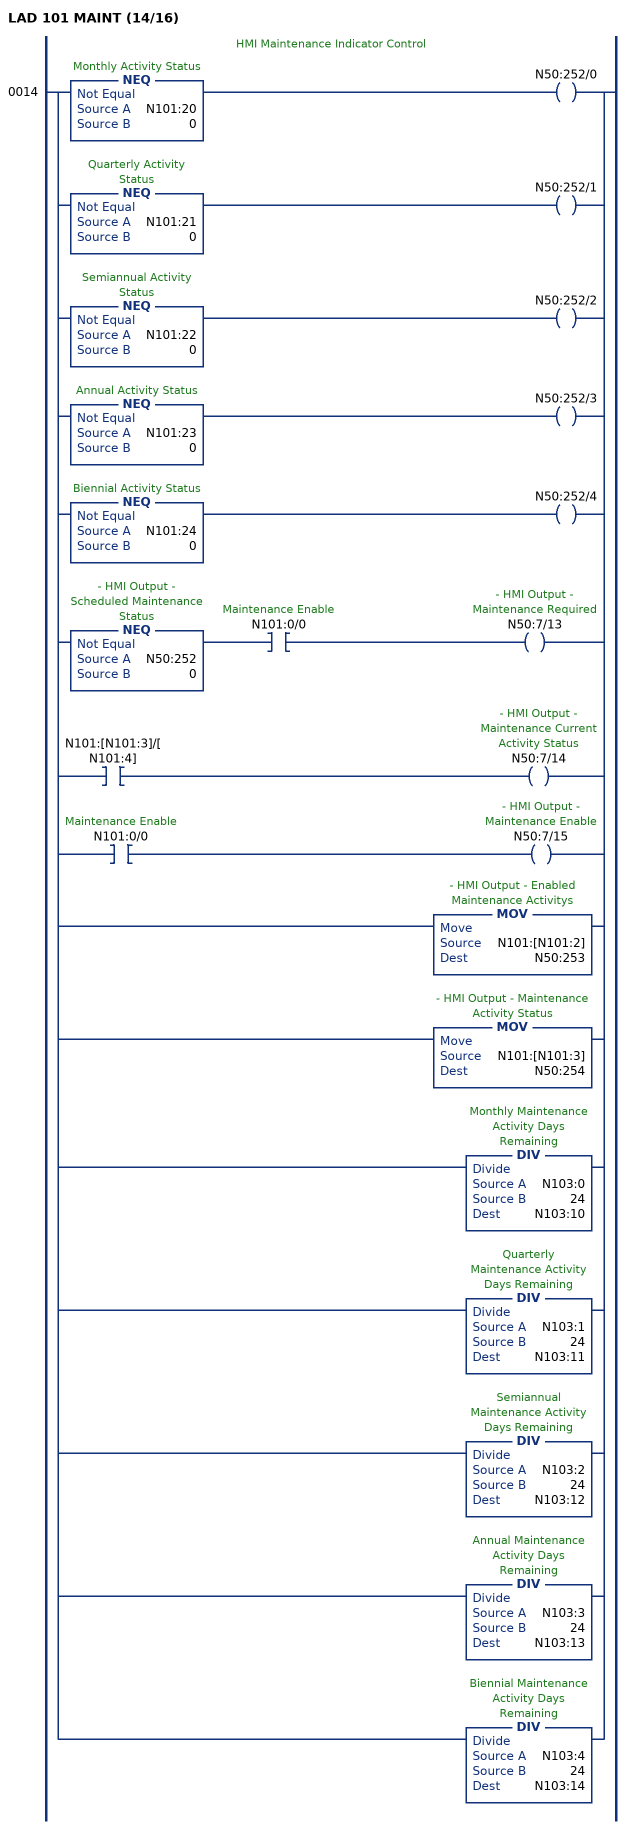
% Rung: 14 %
% HMI Maintenance Indicator Control %
SOR BST BST NEQ N101:20 0 OTE N50:252/0 NXB NEQ N101:21 0 OTE N50:252/1 NXB NEQ N101:22 0 OTE N50:252/2 NXB NEQ N101:23 0 OTE N50:252/3 NXB NEQ N101:24 0 OTE N50:252/4 NXB NEQ N50:252 0 XIC N101:0/0 OTE N50:7/13 BND NXB XIC N101:[N101:3]/[N101:4] OTE N50:7/14 NXB XIC N101:0/0 OTE N50:7/15 NXB BST MOV N101:[N101:2] N50:253 NXB MOV N101:[N101:3] N50:254 BND NXB BST DIV N103:0 24 N103:10 NXB DIV N103:1 24 N103:11 NXB DIV N103:2 24 N103:12 NXB DIV N103:3 24 N103:13 NXB DIV N103:4 24 N103:14 BND BND EOR
%   N101:20  "Monthly Activity Status" %
%   N101:21  "Quarterly Activity Status" %
%   N101:22  "Semiannual Activity Status" %
%   N101:23  "Annual Activity Status" %
%   N101:24  "Biennial Activity Status" %
%   N50:252  "- HMI Output - Scheduled Maintenance Status" %
%   N101:0/0  "Maintenance Enable" %
%   N50:7/13  "- HMI Output - Maintenance Required" %
%   N101:3  "Maintenance Schedule Index Plus 20" %
%   N101:4  "Maintenance Activity Index" %
%   N50:7/14  "- HMI Output - Maintenance Current Activity Status" %
%   N50:7/15  "- HMI Output - Maintenance Enable" %
%   N101:2  "Maintenance Schedule Index Plus 10" %
%   N50:253  "- HMI Output - Enabled Maintenance Activitys" %
%   N50:254  "- HMI Output - Maintenance Activity Status" %
%   N103:0  "Monthly Maintenance Activity Hours Remaining" %
%   N103:10  "Monthly Maintenance Activity Days Remaining" %
%   N103:1  "Quarterly Maintenance Activity Hours Remaining" %
%   N103:11  "Quarterly Maintenance Activity Days Remaining" %
%   N103:2  "Semiannual Maintenance Activity Hours Remaining" %
%   N103:12  "Semiannual Maintenance Activity Days Remaining" %
%   N103:3  "Annual Maintenance Activity Hours Remaining" %
%   N103:13  "Annual Maintenance Activity Days Remaining" %
%   N103:4  "Biennial Maintenance Activity Hours Remaining" %
%   N103:14  "Biennial Maintenance Activity Days Remaining" %

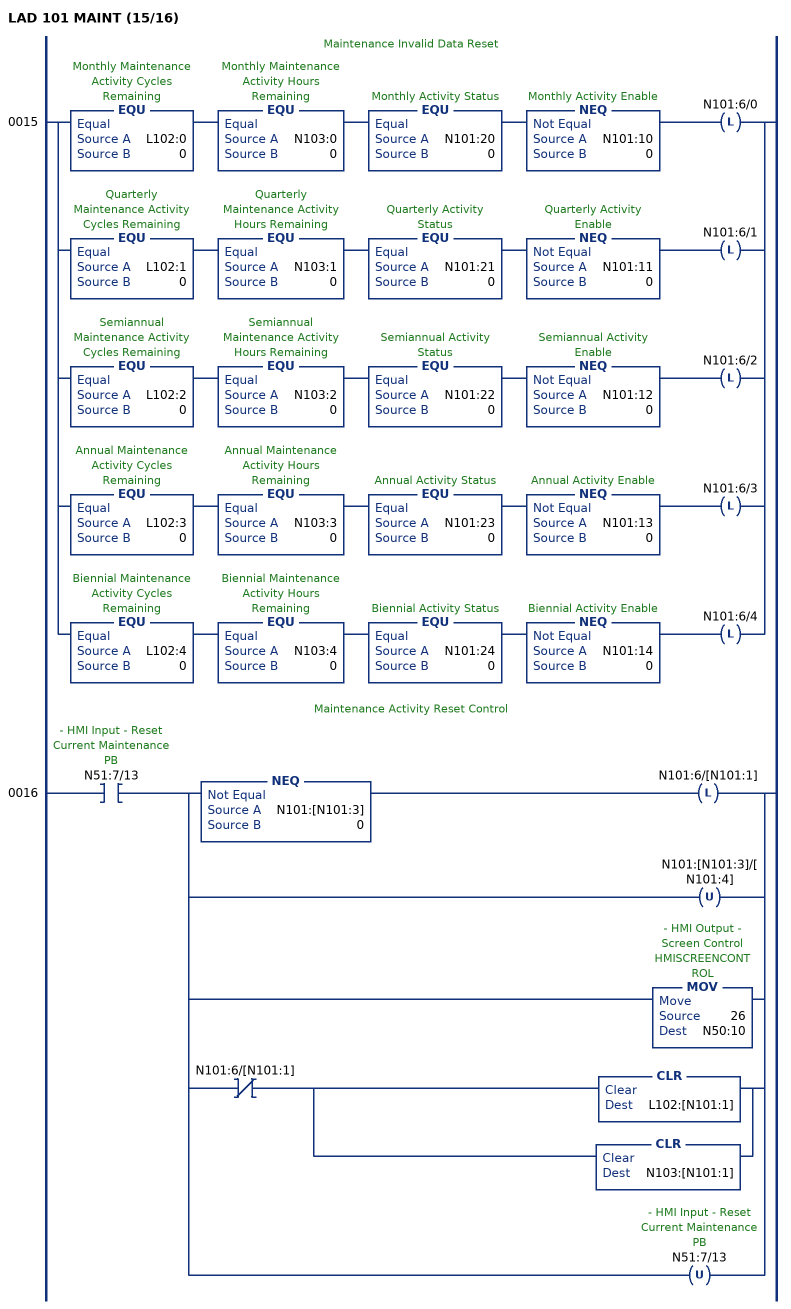
% Rung: 15 %
% Maintenance Invalid Data Reset %
SOR BST EQU L102:0 0 EQU N103:0 0 EQU N101:20 0 NEQ N101:10 0 OTL N101:6/0 NXB EQU L102:1 0 EQU N103:1 0 EQU N101:21 0 NEQ N101:11 0 OTL N101:6/1 NXB EQU L102:2 0 EQU N103:2 0 EQU N101:22 0 NEQ N101:12 0 OTL N101:6/2 NXB EQU L102:3 0 EQU N103:3 0 EQU N101:23 0 NEQ N101:13 0 OTL N101:6/3 NXB EQU L102:4 0 EQU N103:4 0 EQU N101:24 0 NEQ N101:14 0 OTL N101:6/4 BND EOR
%   L102:0  "Monthly Maintenance Activity Cycles Remaining" %
%   N103:0  "Monthly Maintenance Activity Hours Remaining" %
%   N101:20  "Monthly Activity Status" %
%   N101:10  "Monthly Activity Enable" %
%   L102:1  "Quarterly Maintenance Activity Cycles Remaining" %
%   N103:1  "Quarterly Maintenance Activity Hours Remaining" %
%   N101:21  "Quarterly Activity Status" %
%   N101:11  "Quarterly Activity Enable" %
%   L102:2  "Semiannual Maintenance Activity Cycles Remaining" %
%   N103:2  "Semiannual Maintenance Activity Hours Remaining" %
%   N101:22  "Semiannual Activity Status" %
%   N101:12  "Semiannual Activity Enable" %
%   L102:3  "Annual Maintenance Activity Cycles Remaining" %
%   N103:3  "Annual Maintenance Activity Hours Remaining" %
%   N101:23  "Annual Activity Status" %
%   N101:13  "Annual Activity Enable" %
%   L102:4  "Biennial Maintenance Activity Cycles Remaining" %
%   N103:4  "Biennial Maintenance Activity Hours Remaining" %
%   N101:24  "Biennial Activity Status" %
%   N101:14  "Biennial Activity Enable" %
% Rung: 16 %
% Maintenance Activity Reset Control %
SOR XIC N51:7/13 BST NEQ N101:[N101:3] 0 OTL N101:6/[N101:1] NXB OTU N101:[N101:3]/[N101:4] NXB MOV 26 N50:10 NXB XIO N101:6/[N101:1] BST CLR L102:[N101:1] NXB CLR N103:[N101:1] BND NXB OTU N51:7/13 BND EOR
%   N51:7/13  "- HMI Input - Reset Current Maintenance PB" %
%   N101:3  "Maintenance Schedule Index Plus 20" %
%   N101:6  "Maintenance Reset" %
%   N101:1  "Maintenance Schedule Index" %
%   N101:4  "Maintenance Activity Index" %
%   N50:10  HMISCREENCONTROL  "- HMI Output - Screen Control" %

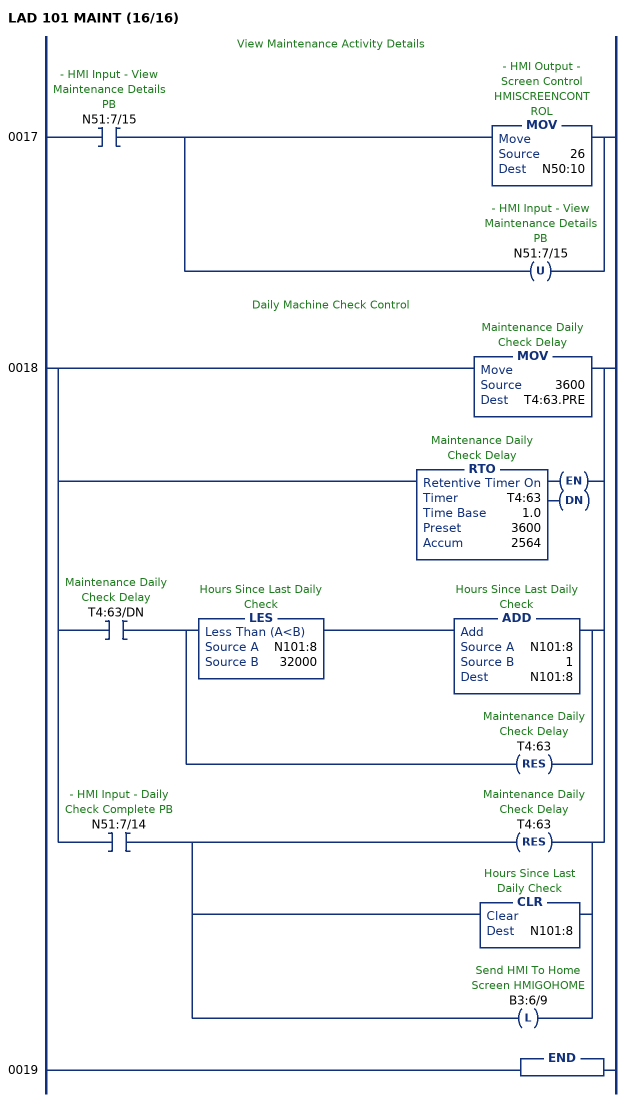
% Rung: 17 %
% View Maintenance Activity Details %
SOR XIC N51:7/15 BST MOV 26 N50:10 NXB OTU N51:7/15 BND EOR
%   N51:7/15  "- HMI Input - View Maintenance Details PB" %
%   N50:10  HMISCREENCONTROL  "- HMI Output - Screen Control" %
% Rung: 18 %
% Daily Machine Check Control %
SOR BST MOV 3600 T4:63.PRE NXB RTO T4:63 1.0 3600 2564 NXB XIC T4:63/DN BST LES N101:8 32000 ADD N101:8 1 N101:8 NXB RES T4:63 BND NXB XIC N51:7/14 BST RES T4:63 NXB CLR N101:8 NXB OTL B3:6/9 BND BND EOR
%   T4:63  "Maintenance Daily Check Delay" %
%   N101:8  "Hours Since Last Daily Check" %
%   N51:7/14  "- HMI Input - Daily Check Complete PB" %
%   B3:6/9  HMIGOHOME  "Send HMI To Home Screen" %
% Rung: 19 %
SOR END EOR

LADDER 115 "PDATA"    % Production Data %
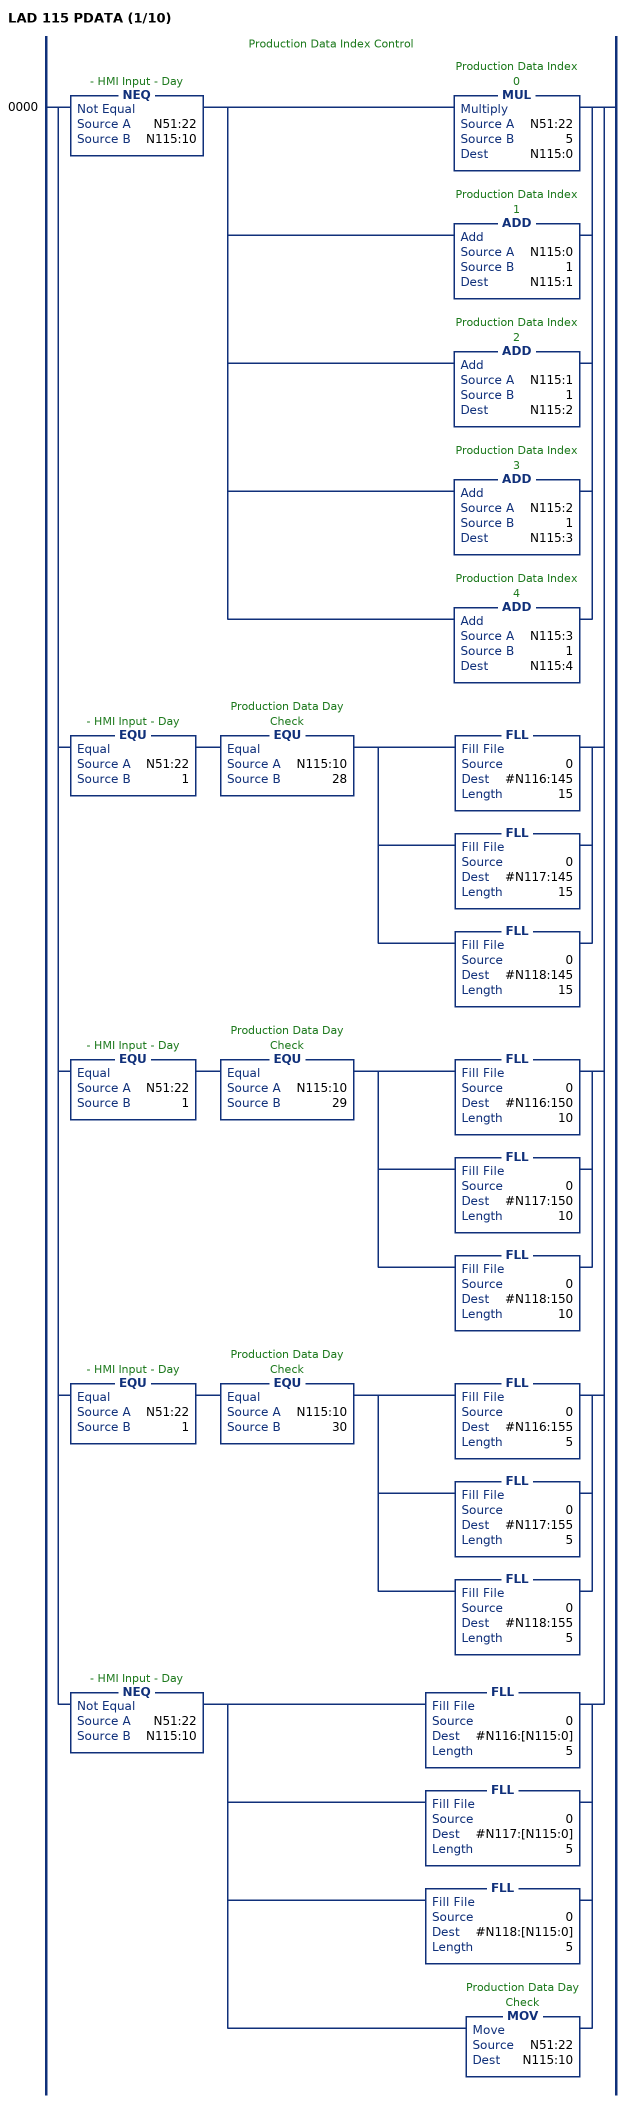
% Rung: 0 %
% Production Data Index Control %
SOR BST NEQ N51:22 N115:10 BST MUL N51:22 5 N115:0 NXB ADD N115:0 1 N115:1 NXB ADD N115:1 1 N115:2 NXB ADD N115:2 1 N115:3 NXB ADD N115:3 1 N115:4 BND NXB EQU N51:22 1 EQU N115:10 28 BST FLL 0 #N116:145 15 NXB FLL 0 #N117:145 15 NXB FLL 0 #N118:145 15 BND NXB EQU N51:22 1 EQU N115:10 29 BST FLL 0 #N116:150 10 NXB FLL 0 #N117:150 10 NXB FLL 0 #N118:150 10 BND NXB EQU N51:22 1 EQU N115:10 30 BST FLL 0 #N116:155 5 NXB FLL 0 #N117:155 5 NXB FLL 0 #N118:155 5 BND NXB NEQ N51:22 N115:10 BST FLL 0 #N116:[N115:0] 5 NXB FLL 0 #N117:[N115:0] 5 NXB FLL 0 #N118:[N115:0] 5 NXB MOV N51:22 N115:10 BND BND EOR
%   N51:22  "- HMI Input - Day" %
%   N115:10  "Production Data Day Check" %
%   N115:0  "Production Data Index 0" %
%   N115:1  "Production Data Index 1" %
%   N115:2  "Production Data Index 2" %
%   N115:3  "Production Data Index 3" %
%   N115:4  "Production Data Index 4" %

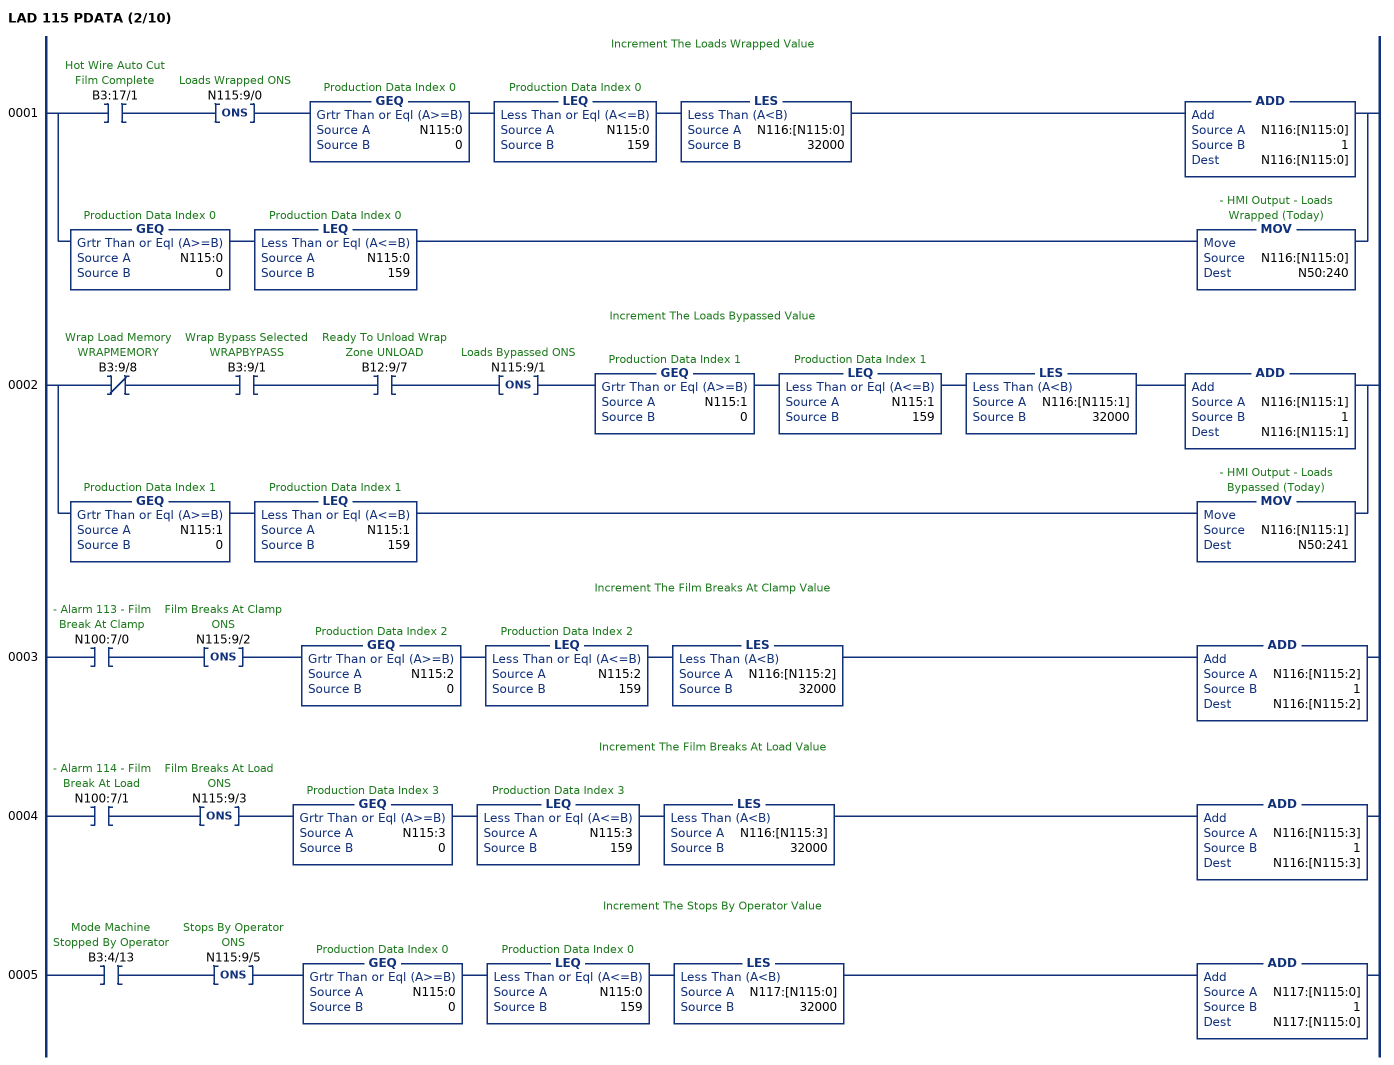
% Rung: 1 %
% Increment The Loads Wrapped Value %
SOR BST XIC B3:17/1 ONS N115:9/0 GEQ N115:0 0 LEQ N115:0 159 LES N116:[N115:0] 32000 ADD N116:[N115:0] 1 N116:[N115:0] NXB GEQ N115:0 0 LEQ N115:0 159 MOV N116:[N115:0] N50:240 BND EOR
%   B3:17/1  "Hot Wire Auto Cut Film Complete" %
%   N115:9/0  "Loads Wrapped ONS" %
%   N115:0  "Production Data Index 0" %
%   N50:240  "- HMI Output - Loads Wrapped (Today)" %
% Rung: 2 %
% Increment The Loads Bypassed Value %
SOR BST XIO B3:9/8 XIC B3:9/1 XIC B12:9/7 ONS N115:9/1 GEQ N115:1 0 LEQ N115:1 159 LES N116:[N115:1] 32000 ADD N116:[N115:1] 1 N116:[N115:1] NXB GEQ N115:1 0 LEQ N115:1 159 MOV N116:[N115:1] N50:241 BND EOR
%   B3:9/8  WRAPMEMORY  "Wrap Load Memory" %
%   B3:9/1  WRAPBYPASS  "Wrap Bypass Selected" %
%   B12:9/7  UNLOAD  "Ready To Unload Wrap Zone" %
%   N115:9/1  "Loads Bypassed ONS" %
%   N115:1  "Production Data Index 1" %
%   N50:241  "- HMI Output - Loads Bypassed (Today)" %
% Rung: 3 %
% Increment The Film Breaks At Clamp Value %
SOR XIC N100:7/0 ONS N115:9/2 GEQ N115:2 0 LEQ N115:2 159 LES N116:[N115:2] 32000 ADD N116:[N115:2] 1 N116:[N115:2] EOR
%   N100:7/0  "- Alarm 113 - Film Break At Clamp" %
%   N115:9/2  "Film Breaks At Clamp ONS" %
%   N115:2  "Production Data Index 2" %
% Rung: 4 %
% Increment The Film Breaks At Load Value %
SOR XIC N100:7/1 ONS N115:9/3 GEQ N115:3 0 LEQ N115:3 159 LES N116:[N115:3] 32000 ADD N116:[N115:3] 1 N116:[N115:3] EOR
%   N100:7/1  "- Alarm 114 - Film Break At Load" %
%   N115:9/3  "Film Breaks At Load ONS" %
%   N115:3  "Production Data Index 3" %
% Rung: 5 %
% Increment The Stops By Operator Value %
SOR XIC B3:4/13 ONS N115:9/5 GEQ N115:0 0 LEQ N115:0 159 LES N117:[N115:0] 32000 ADD N117:[N115:0] 1 N117:[N115:0] EOR
%   B3:4/13  "Mode Machine Stopped By Operator" %
%   N115:9/5  "Stops By Operator ONS" %
%   N115:0  "Production Data Index 0" %

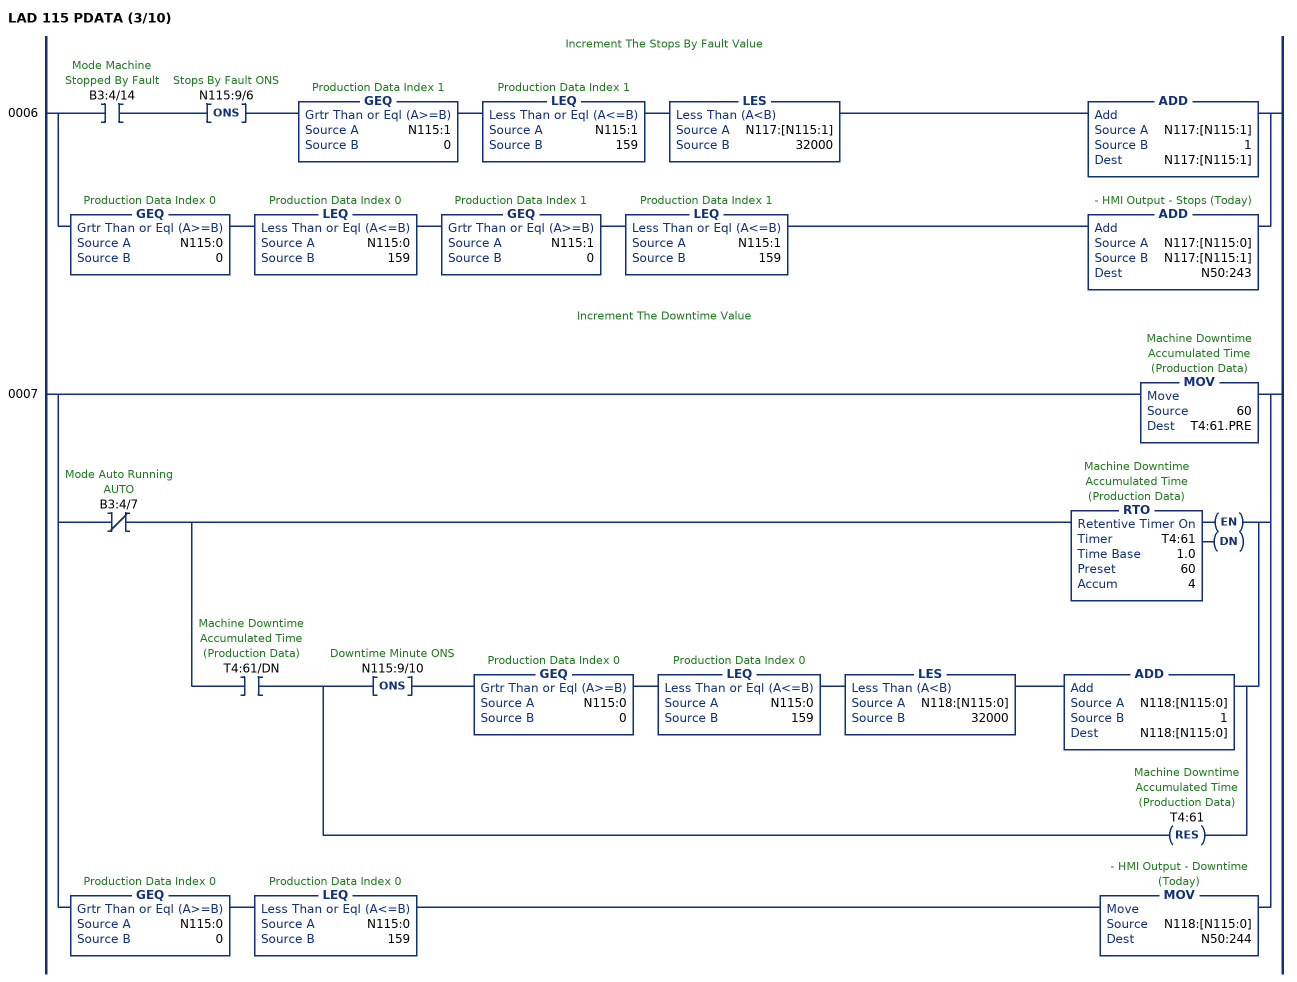
% Rung: 6 %
% Increment The Stops By Fault Value %
SOR BST XIC B3:4/14 ONS N115:9/6 GEQ N115:1 0 LEQ N115:1 159 LES N117:[N115:1] 32000 ADD N117:[N115:1] 1 N117:[N115:1] NXB GEQ N115:0 0 LEQ N115:0 159 GEQ N115:1 0 LEQ N115:1 159 ADD N117:[N115:0] N117:[N115:1] N50:243 BND EOR
%   B3:4/14  "Mode Machine Stopped By Fault" %
%   N115:9/6  "Stops By Fault ONS" %
%   N115:1  "Production Data Index 1" %
%   N115:0  "Production Data Index 0" %
%   N50:243  "- HMI Output - Stops (Today)" %
% Rung: 7 %
% Increment The Downtime Value %
SOR BST MOV 60 T4:61.PRE NXB XIO B3:4/7 BST RTO T4:61 1.0 60 4 NXB XIC T4:61/DN BST ONS N115:9/10 GEQ N115:0 0 LEQ N115:0 159 LES N118:[N115:0] 32000 ADD N118:[N115:0] 1 N118:[N115:0] NXB RES T4:61 BND BND NXB GEQ N115:0 0 LEQ N115:0 159 MOV N118:[N115:0] N50:244 BND EOR
%   T4:61  "Machine Downtime Accumulated Time (Production Data)" %
%   B3:4/7  AUTO  "Mode Auto Running" %
%   N115:9/10  "Downtime Minute ONS" %
%   N115:0  "Production Data Index 0" %
%   N50:244  "- HMI Output - Downtime (Today)" %

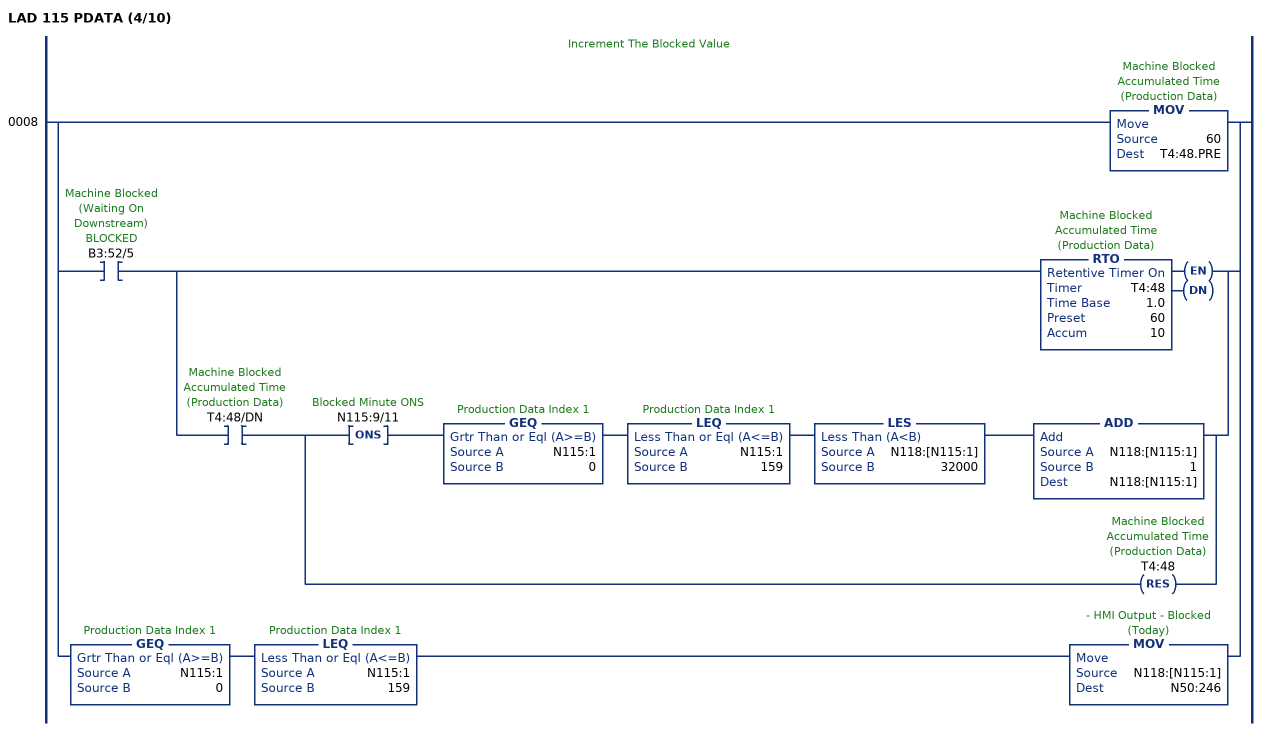
% Rung: 8 %
% Increment The Blocked Value %
SOR BST MOV 60 T4:48.PRE NXB XIC B3:52/5 BST RTO T4:48 1.0 60 10 NXB XIC T4:48/DN BST ONS N115:9/11 GEQ N115:1 0 LEQ N115:1 159 LES N118:[N115:1] 32000 ADD N118:[N115:1] 1 N118:[N115:1] NXB RES T4:48 BND BND NXB GEQ N115:1 0 LEQ N115:1 159 MOV N118:[N115:1] N50:246 BND EOR
%   T4:48  "Machine Blocked Accumulated Time (Production Data)" %
%   B3:52/5  BLOCKED  "Machine Blocked (Waiting On Downstream)" %
%   N115:9/11  "Blocked Minute ONS" %
%   N115:1  "Production Data Index 1" %
%   N50:246  "- HMI Output - Blocked (Today)" %

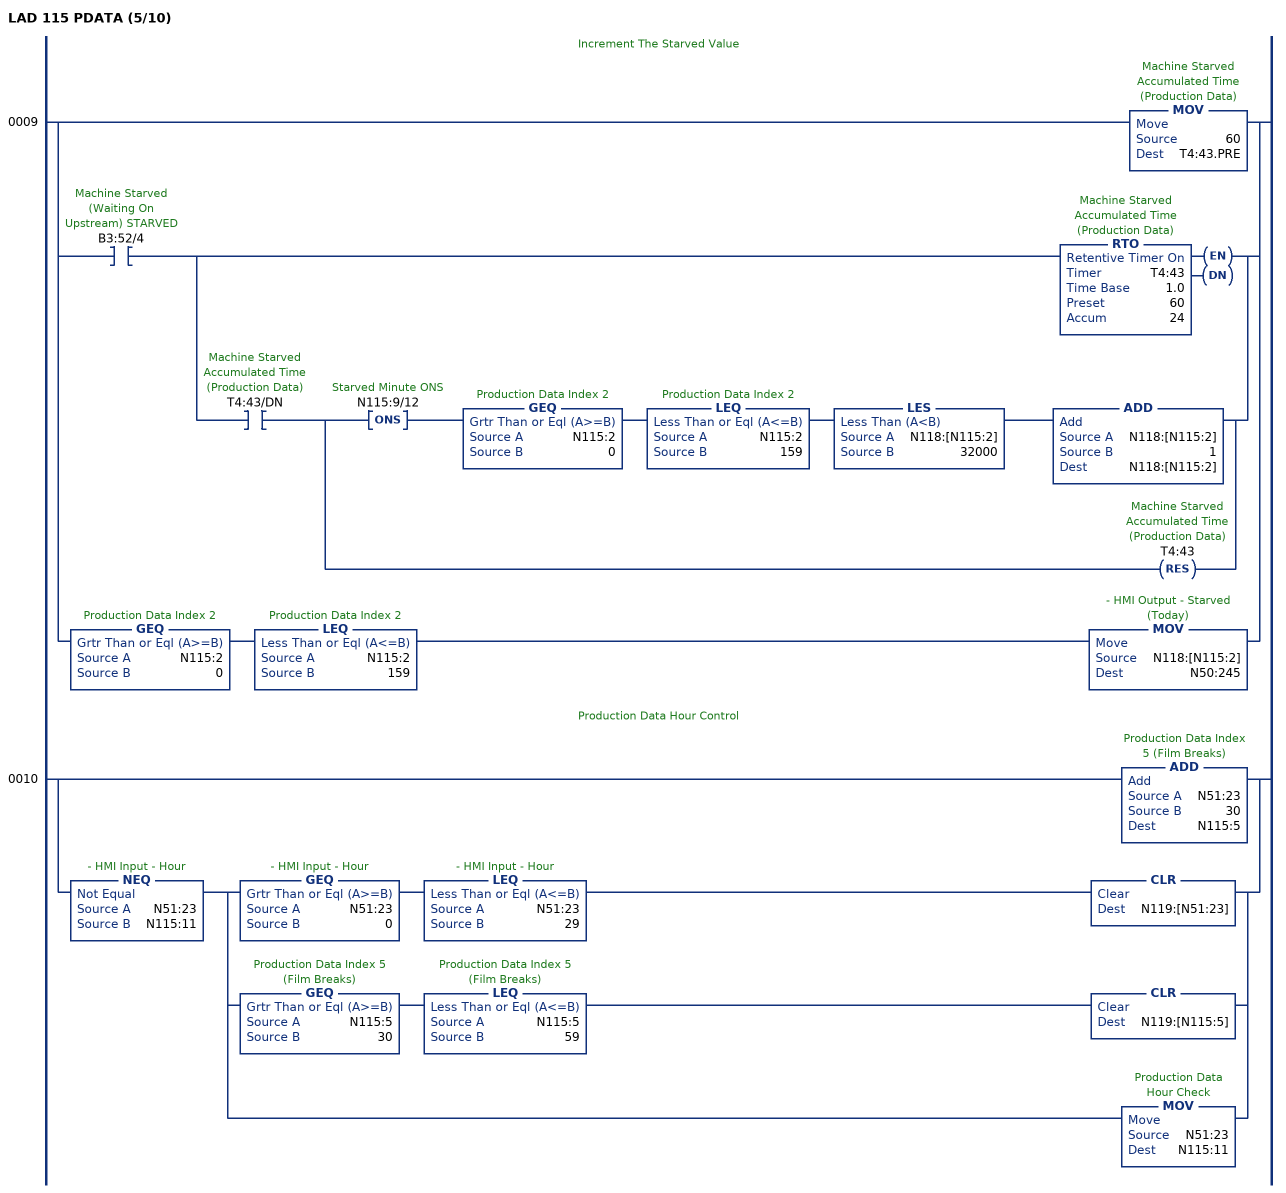
% Rung: 9 %
% Increment The Starved Value %
SOR BST MOV 60 T4:43.PRE NXB XIC B3:52/4 BST RTO T4:43 1.0 60 24 NXB XIC T4:43/DN BST ONS N115:9/12 GEQ N115:2 0 LEQ N115:2 159 LES N118:[N115:2] 32000 ADD N118:[N115:2] 1 N118:[N115:2] NXB RES T4:43 BND BND NXB GEQ N115:2 0 LEQ N115:2 159 MOV N118:[N115:2] N50:245 BND EOR
%   T4:43  "Machine Starved Accumulated Time (Production Data)" %
%   B3:52/4  STARVED  "Machine Starved (Waiting On Upstream)" %
%   N115:9/12  "Starved Minute ONS" %
%   N115:2  "Production Data Index 2" %
%   N50:245  "- HMI Output - Starved (Today)" %
% Rung: 10 %
% Production Data Hour Control %
SOR BST ADD N51:23 30 N115:5 NXB NEQ N51:23 N115:11 BST GEQ N51:23 0 LEQ N51:23 29 CLR N119:[N51:23] NXB GEQ N115:5 30 LEQ N115:5 59 CLR N119:[N115:5] NXB MOV N51:23 N115:11 BND BND EOR
%   N51:23  "- HMI Input - Hour" %
%   N115:5  "Production Data Index 5 (Film Breaks)" %
%   N115:11  "Production Data Hour Check" %

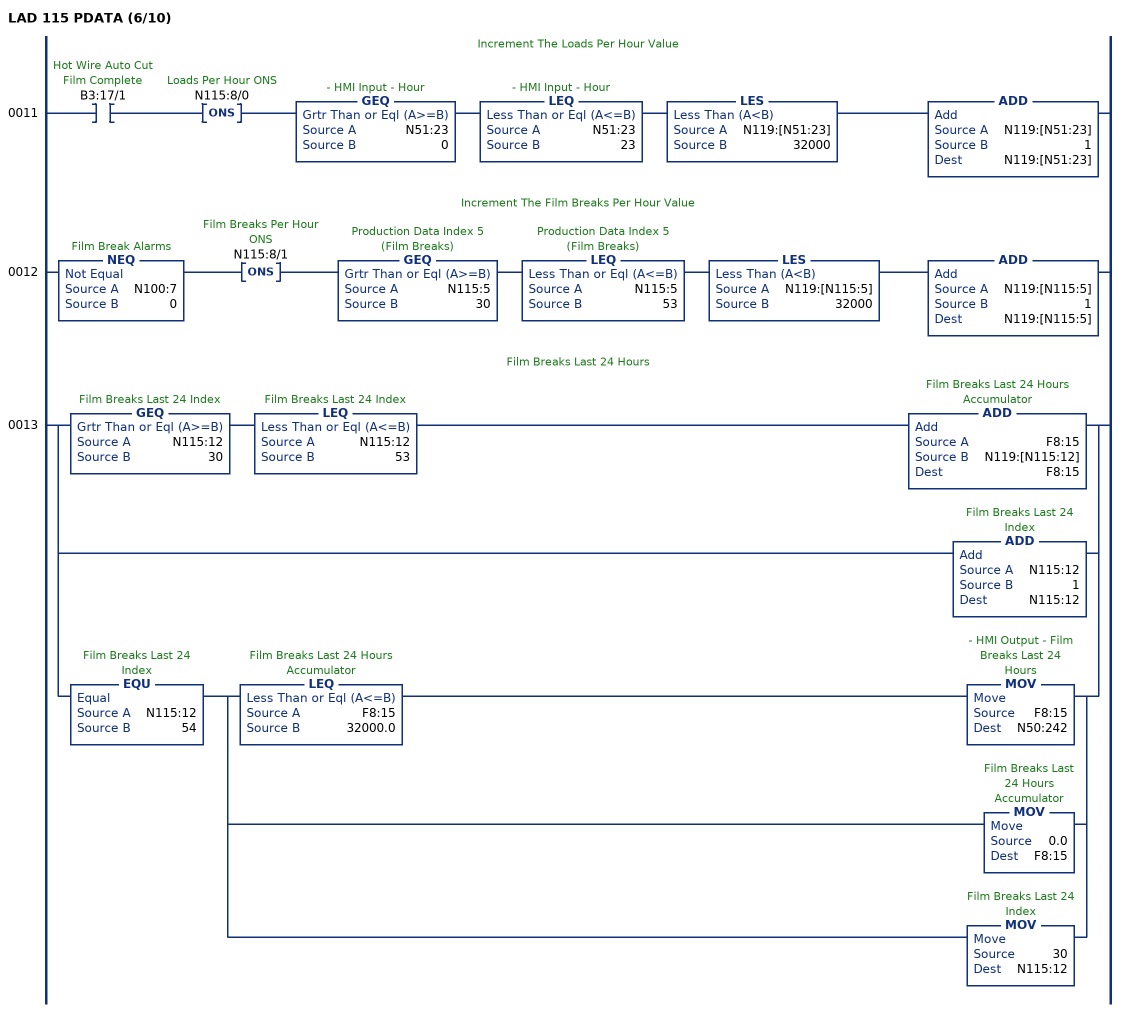
% Rung: 11 %
% Increment The Loads Per Hour Value %
SOR XIC B3:17/1 ONS N115:8/0 GEQ N51:23 0 LEQ N51:23 23 LES N119:[N51:23] 32000 ADD N119:[N51:23] 1 N119:[N51:23] EOR
%   B3:17/1  "Hot Wire Auto Cut Film Complete" %
%   N115:8/0  "Loads Per Hour ONS" %
%   N51:23  "- HMI Input - Hour" %
% Rung: 12 %
% Increment The Film Breaks Per Hour Value %
SOR NEQ N100:7 0 ONS N115:8/1 GEQ N115:5 30 LEQ N115:5 53 LES N119:[N115:5] 32000 ADD N119:[N115:5] 1 N119:[N115:5] EOR
%   N100:7  "Film Break Alarms" %
%   N115:8/1  "Film Breaks Per Hour ONS" %
%   N115:5  "Production Data Index 5 (Film Breaks)" %
% Rung: 13 %
% Film Breaks Last 24 Hours %
SOR BST GEQ N115:12 30 LEQ N115:12 53 ADD F8:15 N119:[N115:12] F8:15 NXB ADD N115:12 1 N115:12 NXB EQU N115:12 54 BST LEQ F8:15 32000.0 MOV F8:15 N50:242 NXB MOV 0.0 F8:15 NXB MOV 30 N115:12 BND BND EOR
%   N115:12  "Film Breaks Last 24 Index" %
%   F8:15  "Film Breaks Last 24 Hours Accumulator" %
%   N50:242  "- HMI Output - Film Breaks Last 24 Hours" %

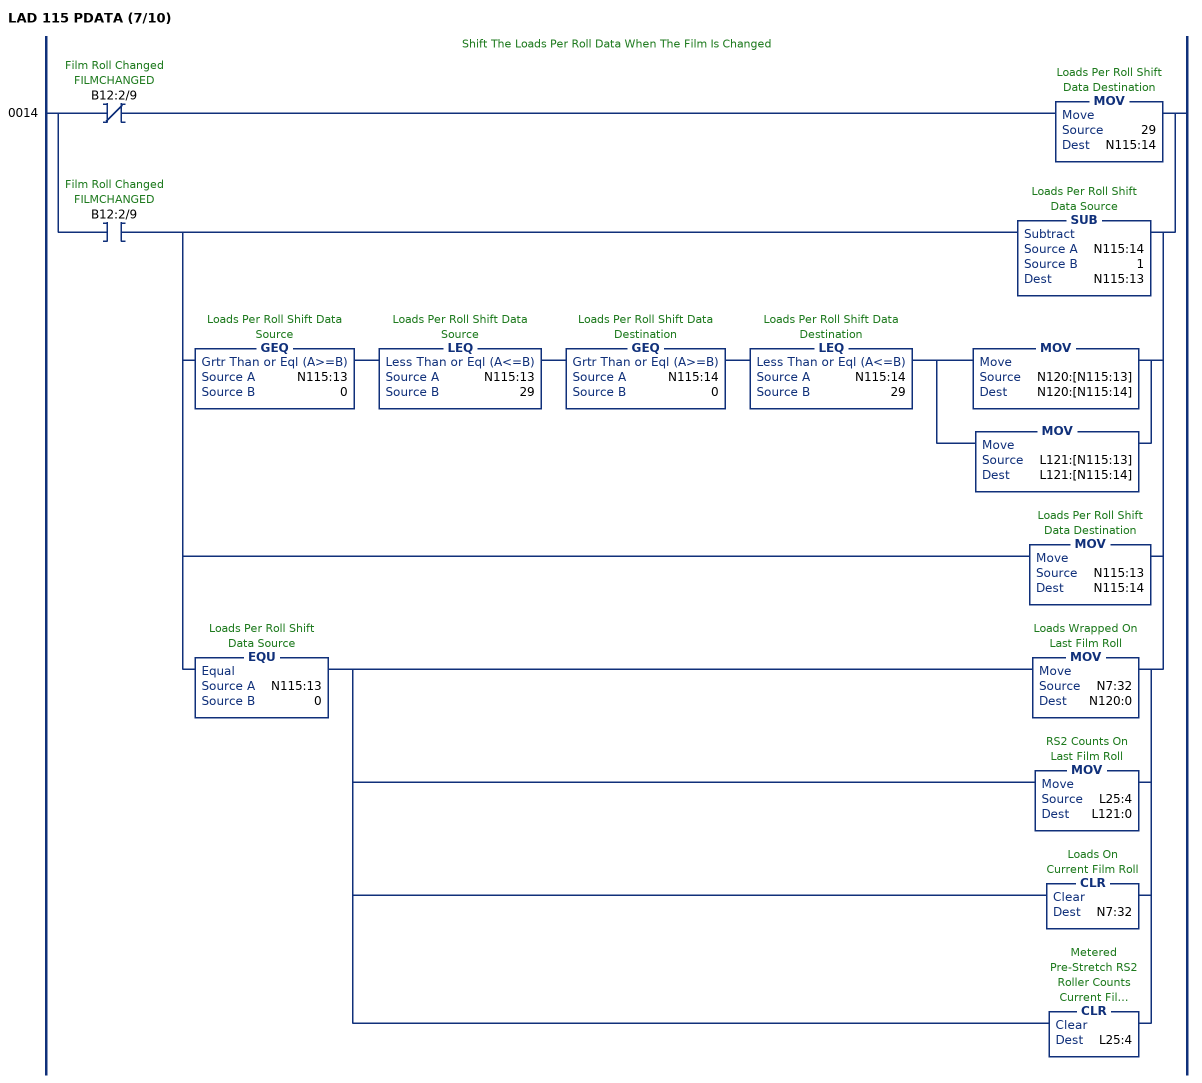
% Rung: 14 %
% Shift The Loads Per Roll Data When The Film Is Changed %
SOR BST XIO B12:2/9 MOV 29 N115:14 NXB XIC B12:2/9 BST SUB N115:14 1 N115:13 NXB GEQ N115:13 0 LEQ N115:13 29 GEQ N115:14 0 LEQ N115:14 29 BST MOV N120:[N115:13] N120:[N115:14] NXB MOV L121:[N115:13] L121:[N115:14] BND NXB MOV N115:13 N115:14 NXB EQU N115:13 0 BST MOV N7:32 N120:0 NXB MOV L25:4 L121:0 NXB CLR N7:32 NXB CLR L25:4 BND BND BND EOR
%   B12:2/9  FILMCHANGED  "Film Roll Changed" %
%   N115:14  "Loads Per Roll Shift Data Destination" %
%   N115:13  "Loads Per Roll Shift Data Source" %
%   N7:32  "Loads On Current Film Roll" %
%   N120:0  "Loads Wrapped On Last Film Roll" %
%   L25:4  "Metered Pre-Stretch RS2 Roller Counts Current Film Roll" %
%   L121:0  "RS2 Counts On Last Film Roll" %

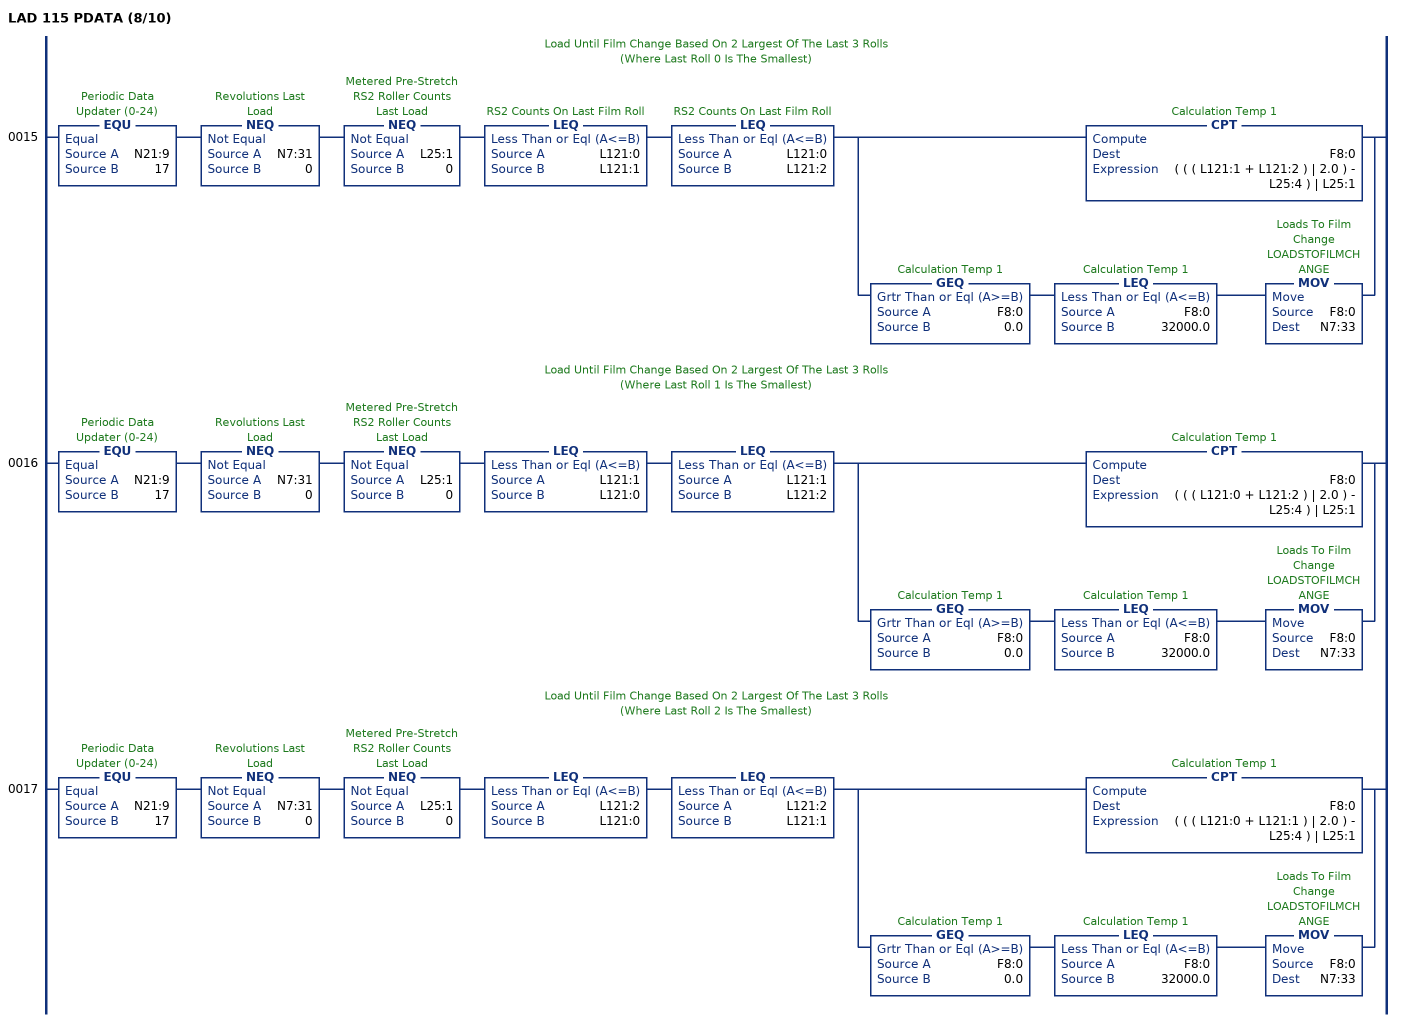
% Rung: 15 %
% Load Until Film Change Based On 2 Largest Of The Last 3 Rolls
% (Where Last Roll 0 Is The Smallest) %
SOR EQU N21:9 17 NEQ N7:31 0 NEQ L25:1 0 LEQ L121:0 L121:1 LEQ L121:0 L121:2 BST CPT F8:0 " ( ( ( L121:1 + L121:2 ) | 2.0 ) - L25:4 ) | L25:1 " NXB GEQ F8:0 0.0 LEQ F8:0 32000.0 MOV F8:0 N7:33 BND EOR
%   N21:9  "Periodic Data Updater (0-24)" %
%   N7:31  "Revolutions Last Load" %
%   L25:1  "Metered Pre-Stretch RS2 Roller Counts Last Load" %
%   L121:0  "RS2 Counts On Last Film Roll" %
%   F8:0  "Calculation Temp 1" %
%   L25:4  "Metered Pre-Stretch RS2 Roller Counts Current Film Roll" %
%   N7:33  LOADSTOFILMCHANGE  "Loads To Film Change" %
% Rung: 16 %
% Load Until Film Change Based On 2 Largest Of The Last 3 Rolls
% (Where Last Roll 1 Is The Smallest) %
SOR EQU N21:9 17 NEQ N7:31 0 NEQ L25:1 0 LEQ L121:1 L121:0 LEQ L121:1 L121:2 BST CPT F8:0 " ( ( ( L121:0 + L121:2 ) | 2.0 ) - L25:4 ) | L25:1 " NXB GEQ F8:0 0.0 LEQ F8:0 32000.0 MOV F8:0 N7:33 BND EOR
%   N21:9  "Periodic Data Updater (0-24)" %
%   N7:31  "Revolutions Last Load" %
%   L25:1  "Metered Pre-Stretch RS2 Roller Counts Last Load" %
%   L121:0  "RS2 Counts On Last Film Roll" %
%   F8:0  "Calculation Temp 1" %
%   L25:4  "Metered Pre-Stretch RS2 Roller Counts Current Film Roll" %
%   N7:33  LOADSTOFILMCHANGE  "Loads To Film Change" %
% Rung: 17 %
% Load Until Film Change Based On 2 Largest Of The Last 3 Rolls
% (Where Last Roll 2 Is The Smallest) %
SOR EQU N21:9 17 NEQ N7:31 0 NEQ L25:1 0 LEQ L121:2 L121:0 LEQ L121:2 L121:1 BST CPT F8:0 " ( ( ( L121:0 + L121:1 ) | 2.0 ) - L25:4 ) | L25:1 " NXB GEQ F8:0 0.0 LEQ F8:0 32000.0 MOV F8:0 N7:33 BND EOR
%   N21:9  "Periodic Data Updater (0-24)" %
%   N7:31  "Revolutions Last Load" %
%   L25:1  "Metered Pre-Stretch RS2 Roller Counts Last Load" %
%   L121:0  "RS2 Counts On Last Film Roll" %
%   F8:0  "Calculation Temp 1" %
%   L25:4  "Metered Pre-Stretch RS2 Roller Counts Current Film Roll" %
%   N7:33  LOADSTOFILMCHANGE  "Loads To Film Change" %

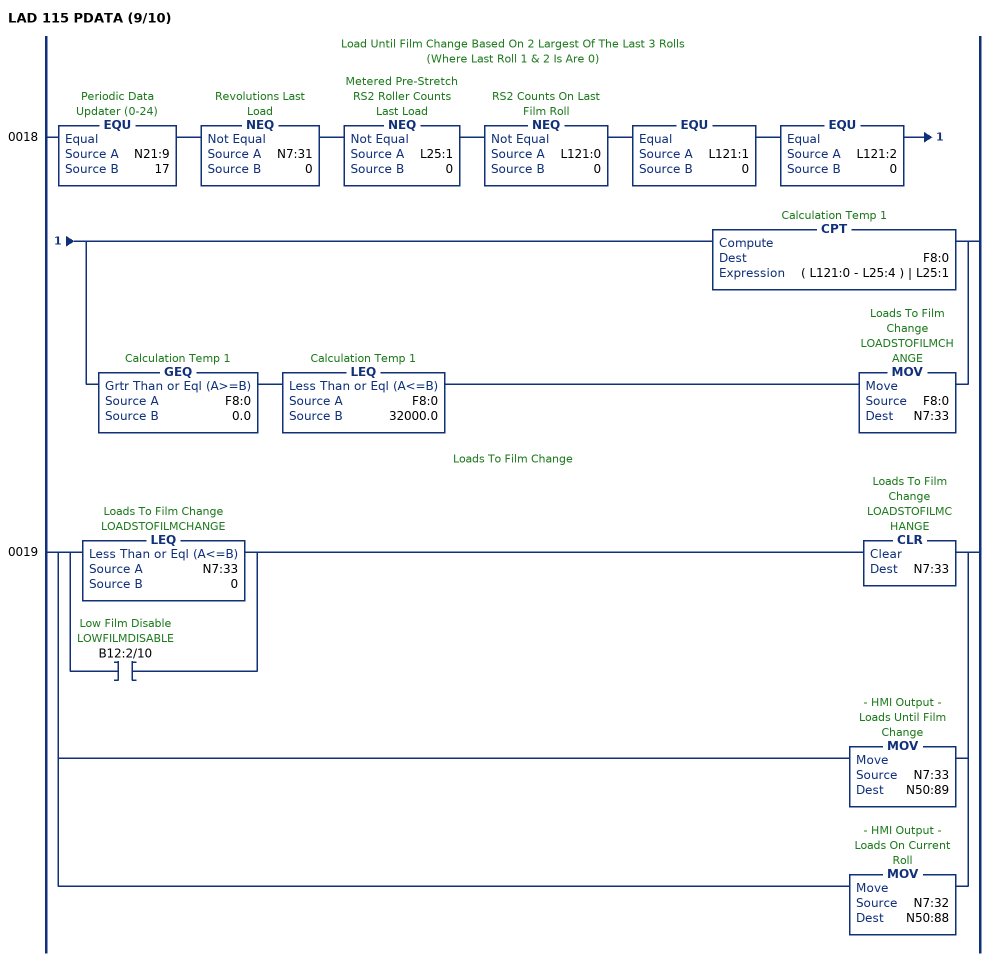
% Rung: 18 %
% Load Until Film Change Based On 2 Largest Of The Last 3 Rolls
% (Where Last Roll 1 & 2 Is Are 0) %
SOR EQU N21:9 17 NEQ N7:31 0 NEQ L25:1 0 NEQ L121:0 0 EQU L121:1 0 EQU L121:2 0 BST CPT F8:0 " ( L121:0 - L25:4 ) | L25:1 " NXB GEQ F8:0 0.0 LEQ F8:0 32000.0 MOV F8:0 N7:33 BND EOR
%   N21:9  "Periodic Data Updater (0-24)" %
%   N7:31  "Revolutions Last Load" %
%   L25:1  "Metered Pre-Stretch RS2 Roller Counts Last Load" %
%   L121:0  "RS2 Counts On Last Film Roll" %
%   F8:0  "Calculation Temp 1" %
%   L25:4  "Metered Pre-Stretch RS2 Roller Counts Current Film Roll" %
%   N7:33  LOADSTOFILMCHANGE  "Loads To Film Change" %
% Rung: 19 %
% Loads To Film Change %
SOR BST BST LEQ N7:33 0 NXB XIC B12:2/10 BND CLR N7:33 NXB MOV N7:33 N50:89 NXB MOV N7:32 N50:88 BND EOR
%   N7:33  LOADSTOFILMCHANGE  "Loads To Film Change" %
%   B12:2/10  LOWFILMDISABLE  "Low Film Disable" %
%   N50:89  "- HMI Output - Loads Until Film Change" %
%   N7:32  "Loads On Current Film Roll" %
%   N50:88  "- HMI Output - Loads On Current Roll" %

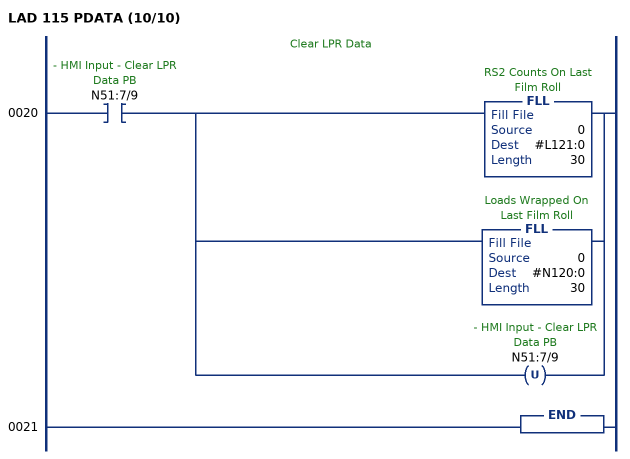
% Rung: 20 %
% Clear LPR Data %
SOR XIC N51:7/9 BST FLL 0 #L121:0 30 NXB FLL 0 #N120:0 30 NXB OTU N51:7/9 BND EOR
%   N51:7/9  "- HMI Input - Clear LPR Data PB" %
%   L121:0  "RS2 Counts On Last Film Roll" %
%   N120:0  "Loads Wrapped On Last Film Roll" %
% Rung: 21 %
SOR END EOR

LADDER 116 "PCHART"    % Production Chart %
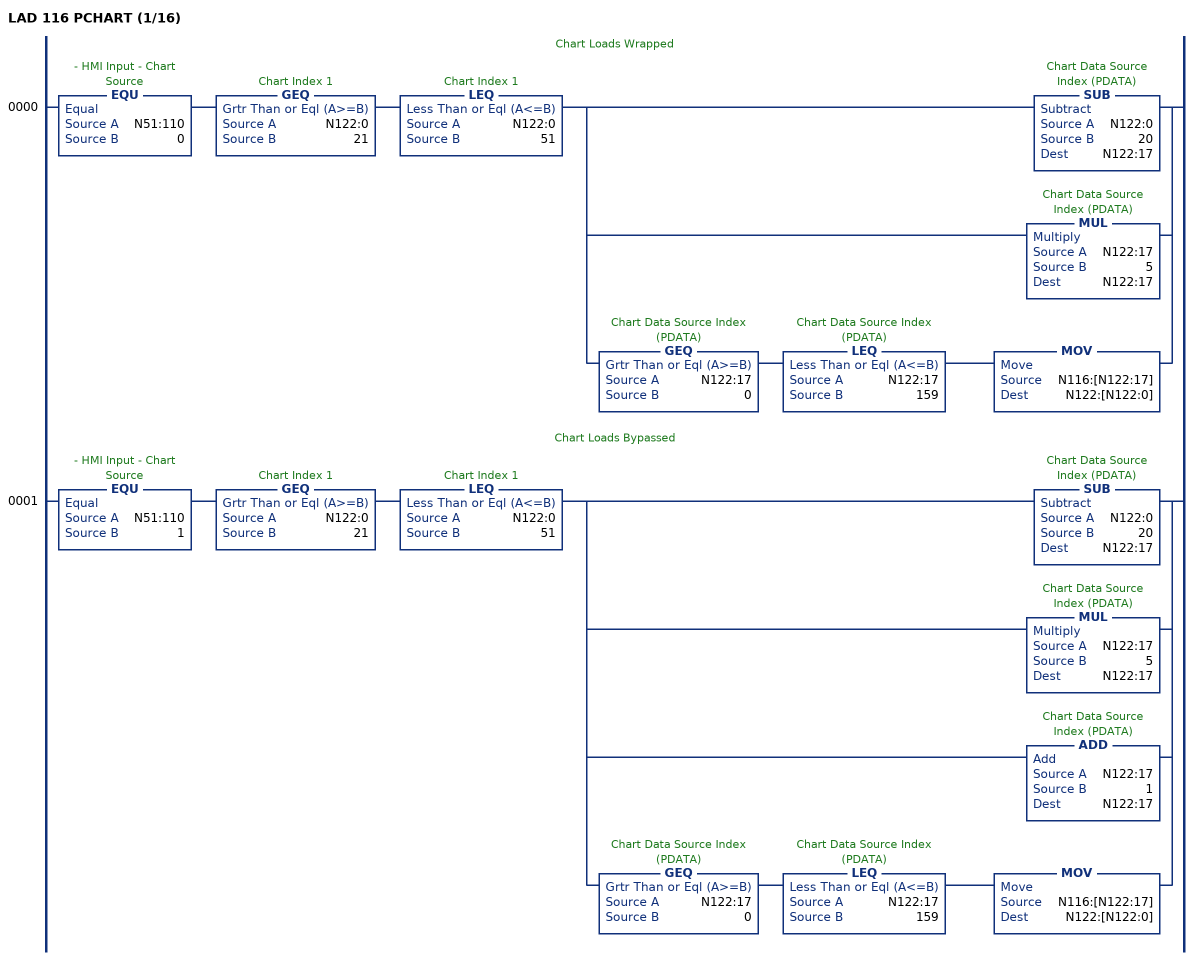
% Rung: 0 %
% Chart Loads Wrapped %
SOR EQU N51:110 0 GEQ N122:0 21 LEQ N122:0 51 BST SUB N122:0 20 N122:17 NXB MUL N122:17 5 N122:17 NXB GEQ N122:17 0 LEQ N122:17 159 MOV N116:[N122:17] N122:[N122:0] BND EOR
%   N51:110  "- HMI Input - Chart Source" %
%   N122:0  "Chart Index 1" %
%   N122:17  "Chart Data Source Index (PDATA)" %
% Rung: 1 %
% Chart Loads Bypassed %
SOR EQU N51:110 1 GEQ N122:0 21 LEQ N122:0 51 BST SUB N122:0 20 N122:17 NXB MUL N122:17 5 N122:17 NXB ADD N122:17 1 N122:17 NXB GEQ N122:17 0 LEQ N122:17 159 MOV N116:[N122:17] N122:[N122:0] BND EOR
%   N51:110  "- HMI Input - Chart Source" %
%   N122:0  "Chart Index 1" %
%   N122:17  "Chart Data Source Index (PDATA)" %

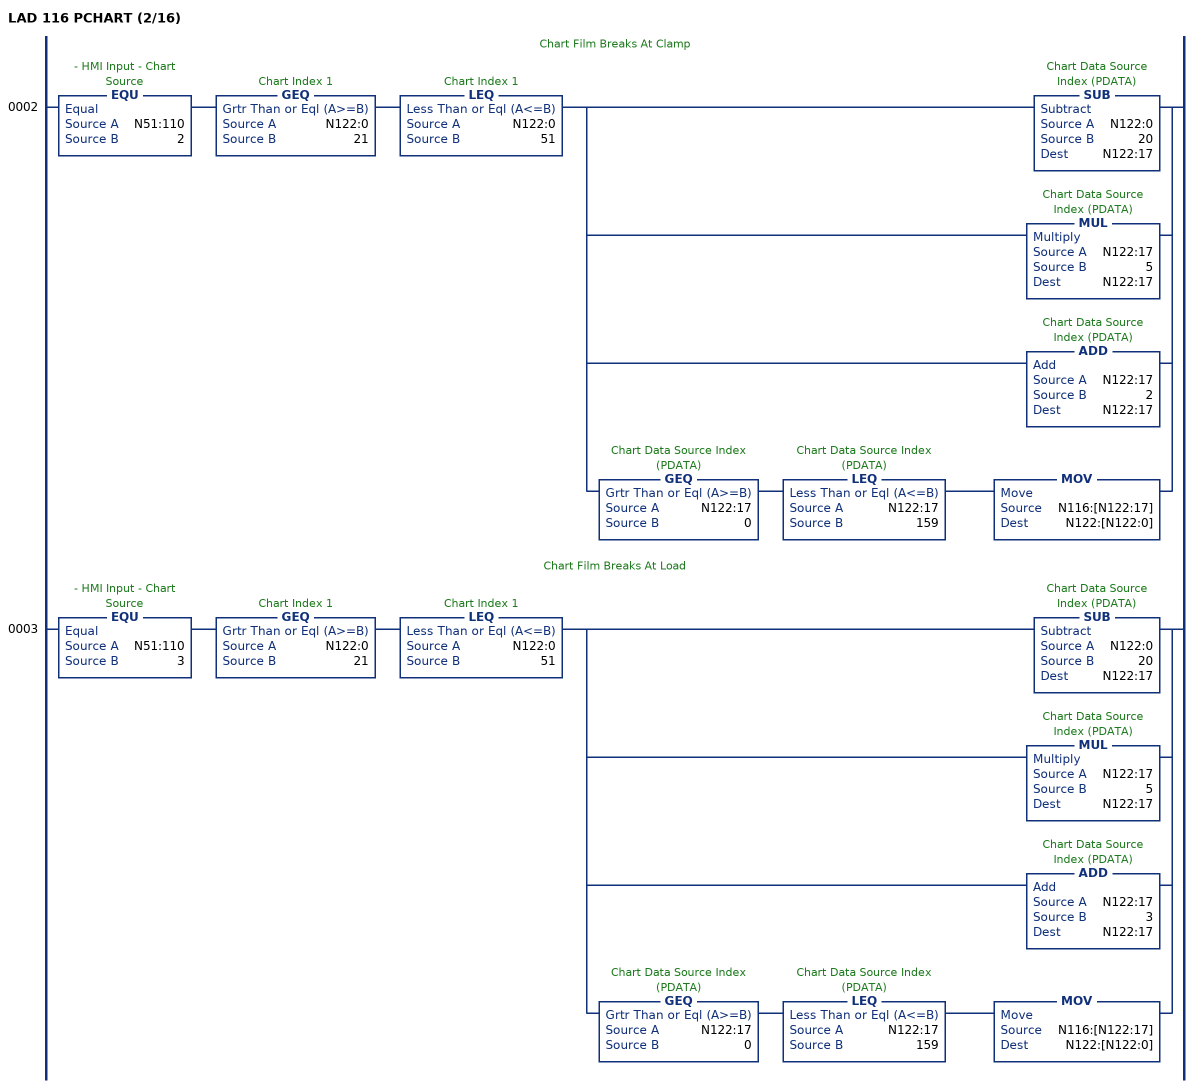
% Rung: 2 %
% Chart Film Breaks At Clamp %
SOR EQU N51:110 2 GEQ N122:0 21 LEQ N122:0 51 BST SUB N122:0 20 N122:17 NXB MUL N122:17 5 N122:17 NXB ADD N122:17 2 N122:17 NXB GEQ N122:17 0 LEQ N122:17 159 MOV N116:[N122:17] N122:[N122:0] BND EOR
%   N51:110  "- HMI Input - Chart Source" %
%   N122:0  "Chart Index 1" %
%   N122:17  "Chart Data Source Index (PDATA)" %
% Rung: 3 %
% Chart Film Breaks At Load %
SOR EQU N51:110 3 GEQ N122:0 21 LEQ N122:0 51 BST SUB N122:0 20 N122:17 NXB MUL N122:17 5 N122:17 NXB ADD N122:17 3 N122:17 NXB GEQ N122:17 0 LEQ N122:17 159 MOV N116:[N122:17] N122:[N122:0] BND EOR
%   N51:110  "- HMI Input - Chart Source" %
%   N122:0  "Chart Index 1" %
%   N122:17  "Chart Data Source Index (PDATA)" %

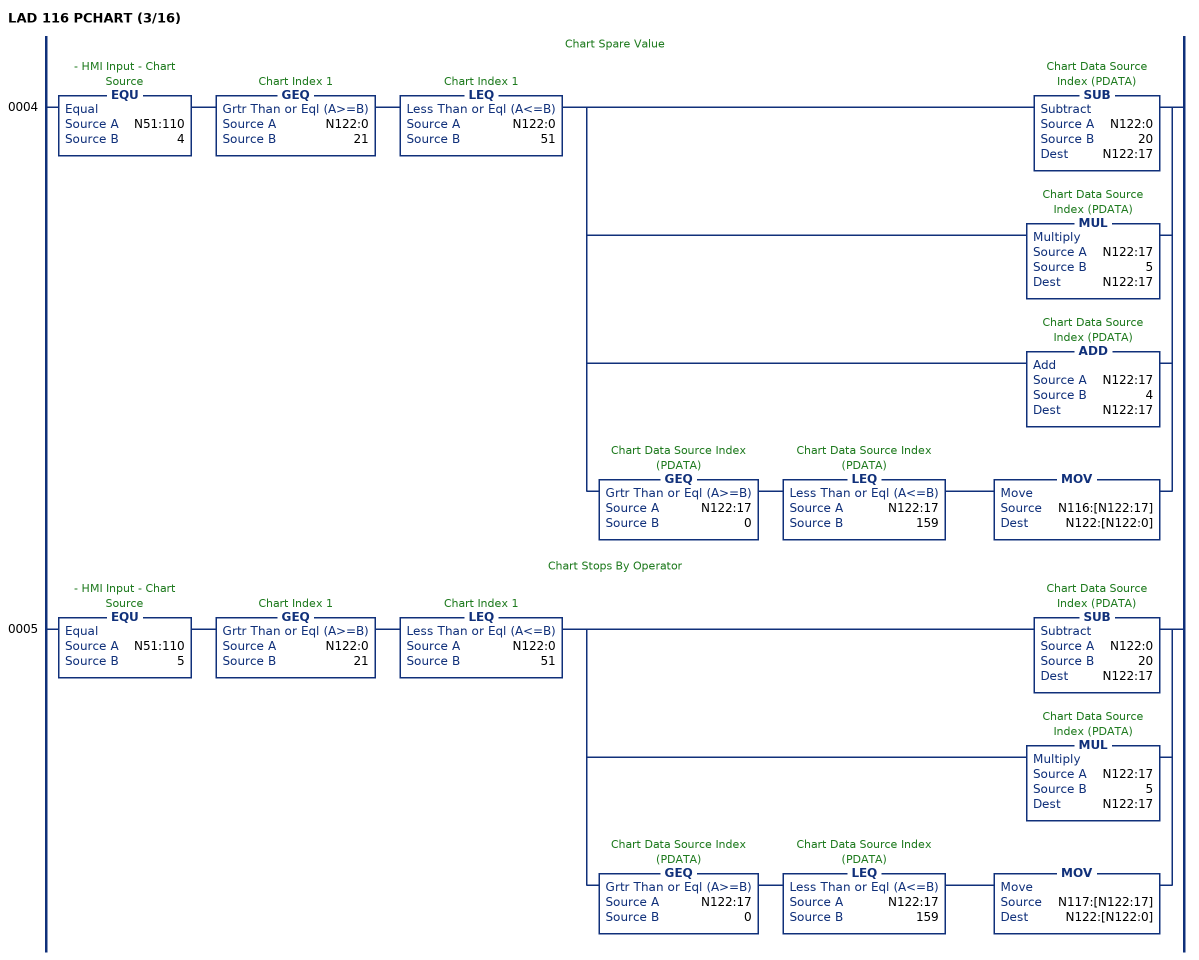
% Rung: 4 %
% Chart Spare Value %
SOR EQU N51:110 4 GEQ N122:0 21 LEQ N122:0 51 BST SUB N122:0 20 N122:17 NXB MUL N122:17 5 N122:17 NXB ADD N122:17 4 N122:17 NXB GEQ N122:17 0 LEQ N122:17 159 MOV N116:[N122:17] N122:[N122:0] BND EOR
%   N51:110  "- HMI Input - Chart Source" %
%   N122:0  "Chart Index 1" %
%   N122:17  "Chart Data Source Index (PDATA)" %
% Rung: 5 %
% Chart Stops By Operator %
SOR EQU N51:110 5 GEQ N122:0 21 LEQ N122:0 51 BST SUB N122:0 20 N122:17 NXB MUL N122:17 5 N122:17 NXB GEQ N122:17 0 LEQ N122:17 159 MOV N117:[N122:17] N122:[N122:0] BND EOR
%   N51:110  "- HMI Input - Chart Source" %
%   N122:0  "Chart Index 1" %
%   N122:17  "Chart Data Source Index (PDATA)" %

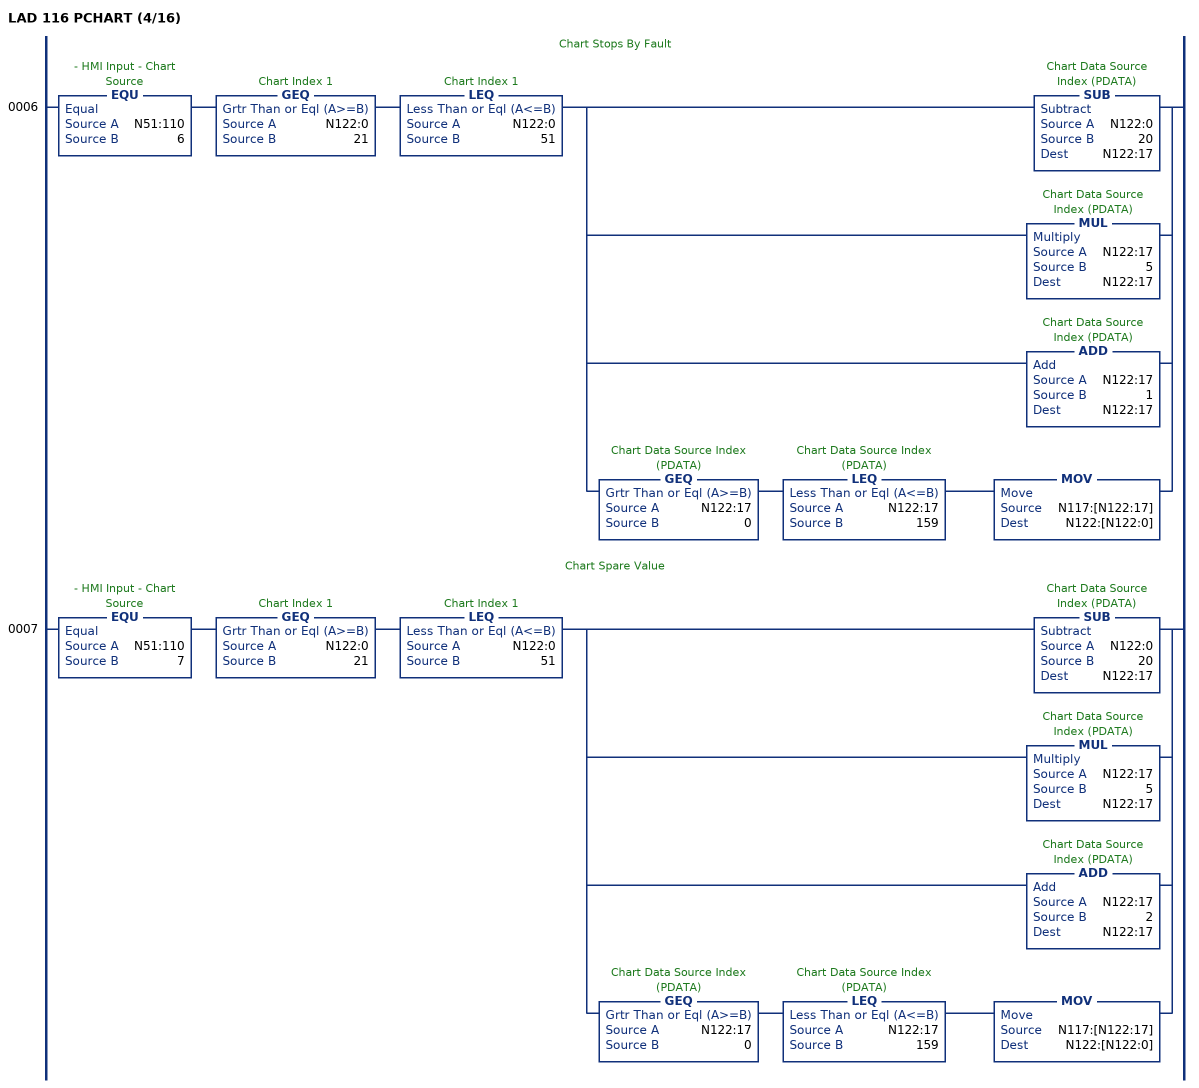
% Rung: 6 %
% Chart Stops By Fault %
SOR EQU N51:110 6 GEQ N122:0 21 LEQ N122:0 51 BST SUB N122:0 20 N122:17 NXB MUL N122:17 5 N122:17 NXB ADD N122:17 1 N122:17 NXB GEQ N122:17 0 LEQ N122:17 159 MOV N117:[N122:17] N122:[N122:0] BND EOR
%   N51:110  "- HMI Input - Chart Source" %
%   N122:0  "Chart Index 1" %
%   N122:17  "Chart Data Source Index (PDATA)" %
% Rung: 7 %
% Chart Spare Value %
SOR EQU N51:110 7 GEQ N122:0 21 LEQ N122:0 51 BST SUB N122:0 20 N122:17 NXB MUL N122:17 5 N122:17 NXB ADD N122:17 2 N122:17 NXB GEQ N122:17 0 LEQ N122:17 159 MOV N117:[N122:17] N122:[N122:0] BND EOR
%   N51:110  "- HMI Input - Chart Source" %
%   N122:0  "Chart Index 1" %
%   N122:17  "Chart Data Source Index (PDATA)" %

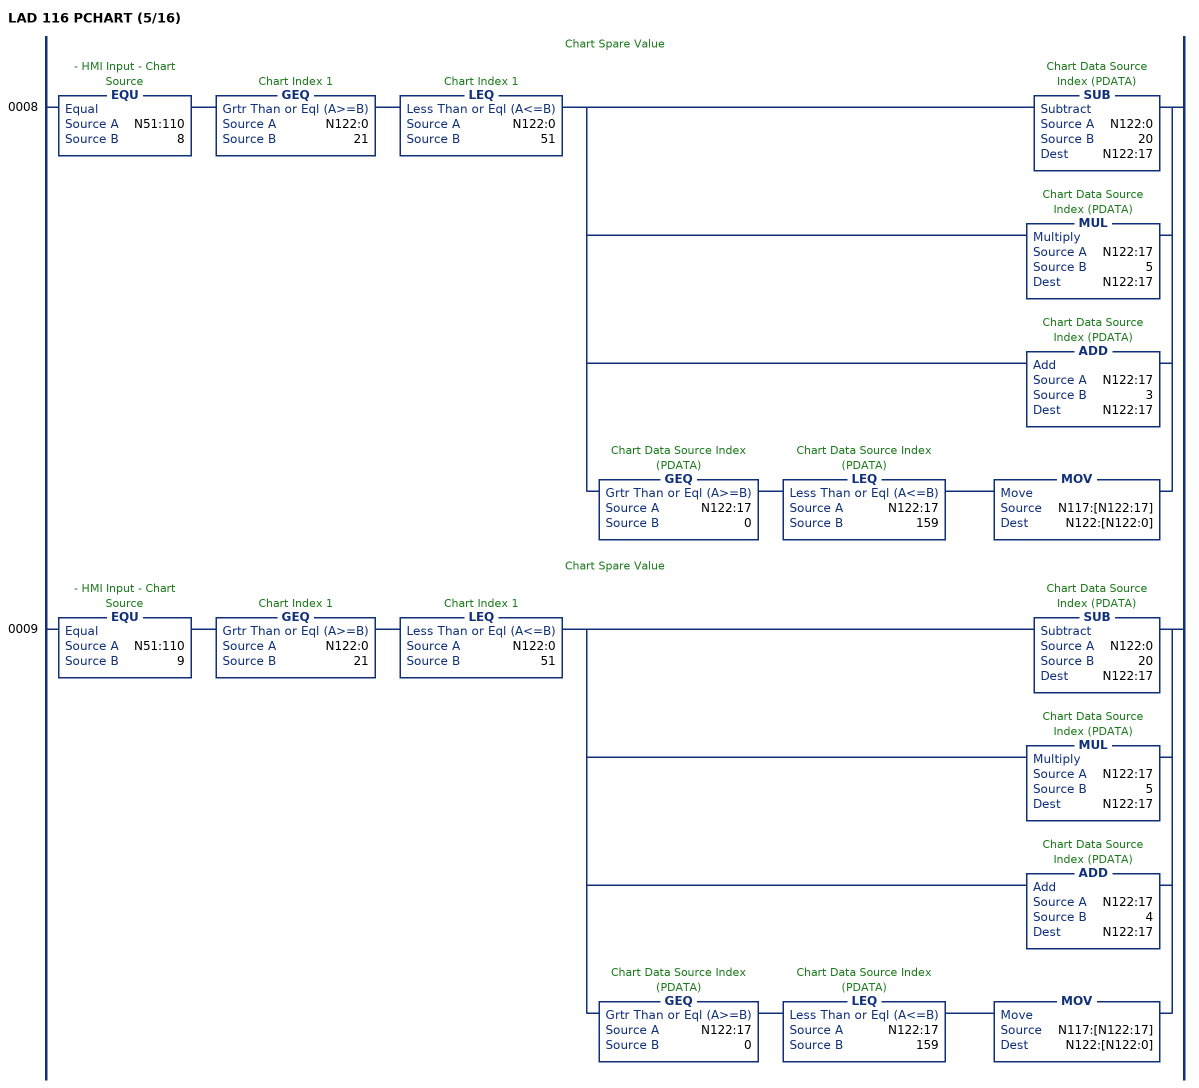
% Rung: 8 %
% Chart Spare Value %
SOR EQU N51:110 8 GEQ N122:0 21 LEQ N122:0 51 BST SUB N122:0 20 N122:17 NXB MUL N122:17 5 N122:17 NXB ADD N122:17 3 N122:17 NXB GEQ N122:17 0 LEQ N122:17 159 MOV N117:[N122:17] N122:[N122:0] BND EOR
%   N51:110  "- HMI Input - Chart Source" %
%   N122:0  "Chart Index 1" %
%   N122:17  "Chart Data Source Index (PDATA)" %
% Rung: 9 %
% Chart Spare Value %
SOR EQU N51:110 9 GEQ N122:0 21 LEQ N122:0 51 BST SUB N122:0 20 N122:17 NXB MUL N122:17 5 N122:17 NXB ADD N122:17 4 N122:17 NXB GEQ N122:17 0 LEQ N122:17 159 MOV N117:[N122:17] N122:[N122:0] BND EOR
%   N51:110  "- HMI Input - Chart Source" %
%   N122:0  "Chart Index 1" %
%   N122:17  "Chart Data Source Index (PDATA)" %

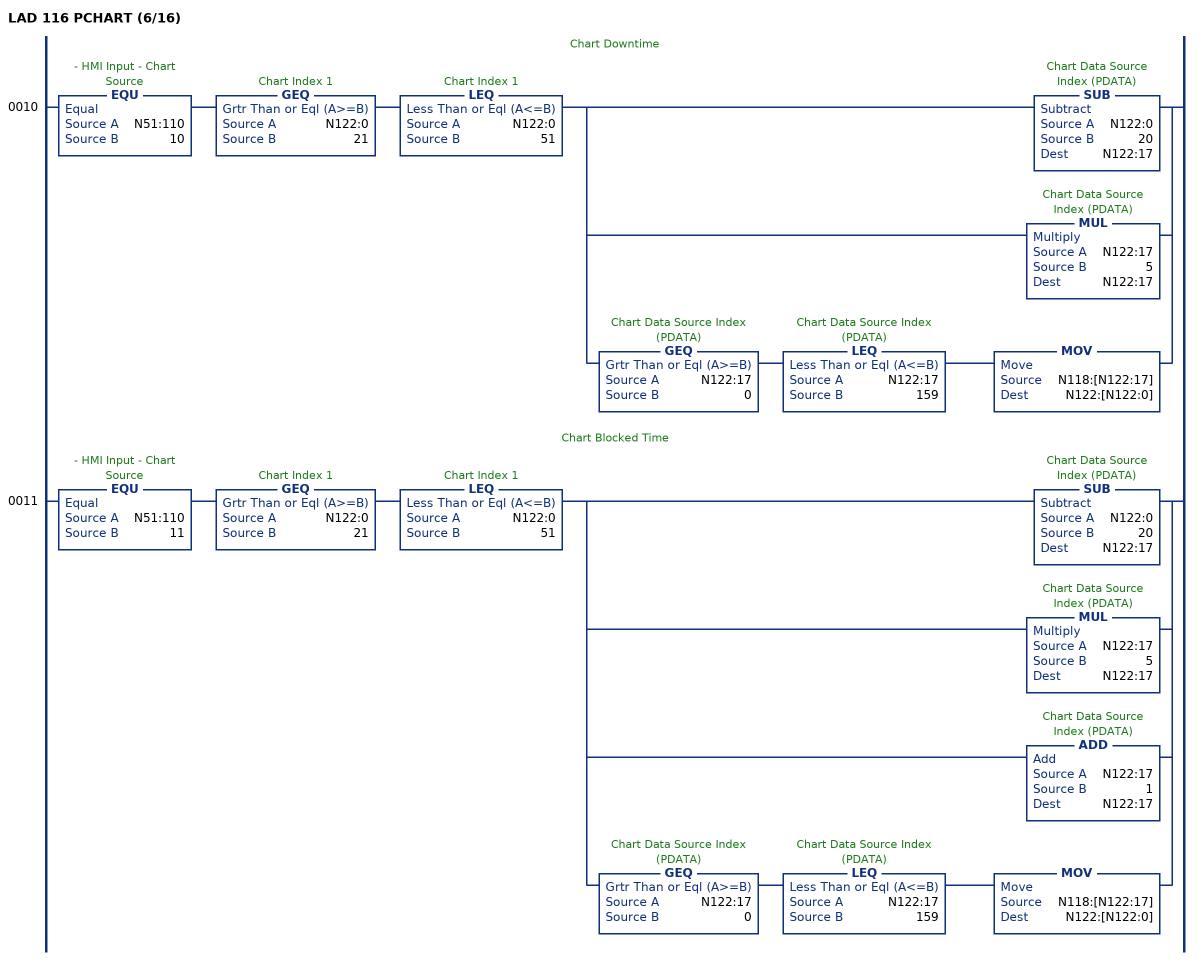
% Rung: 10 %
% Chart Downtime %
SOR EQU N51:110 10 GEQ N122:0 21 LEQ N122:0 51 BST SUB N122:0 20 N122:17 NXB MUL N122:17 5 N122:17 NXB GEQ N122:17 0 LEQ N122:17 159 MOV N118:[N122:17] N122:[N122:0] BND EOR
%   N51:110  "- HMI Input - Chart Source" %
%   N122:0  "Chart Index 1" %
%   N122:17  "Chart Data Source Index (PDATA)" %
% Rung: 11 %
% Chart Blocked Time %
SOR EQU N51:110 11 GEQ N122:0 21 LEQ N122:0 51 BST SUB N122:0 20 N122:17 NXB MUL N122:17 5 N122:17 NXB ADD N122:17 1 N122:17 NXB GEQ N122:17 0 LEQ N122:17 159 MOV N118:[N122:17] N122:[N122:0] BND EOR
%   N51:110  "- HMI Input - Chart Source" %
%   N122:0  "Chart Index 1" %
%   N122:17  "Chart Data Source Index (PDATA)" %

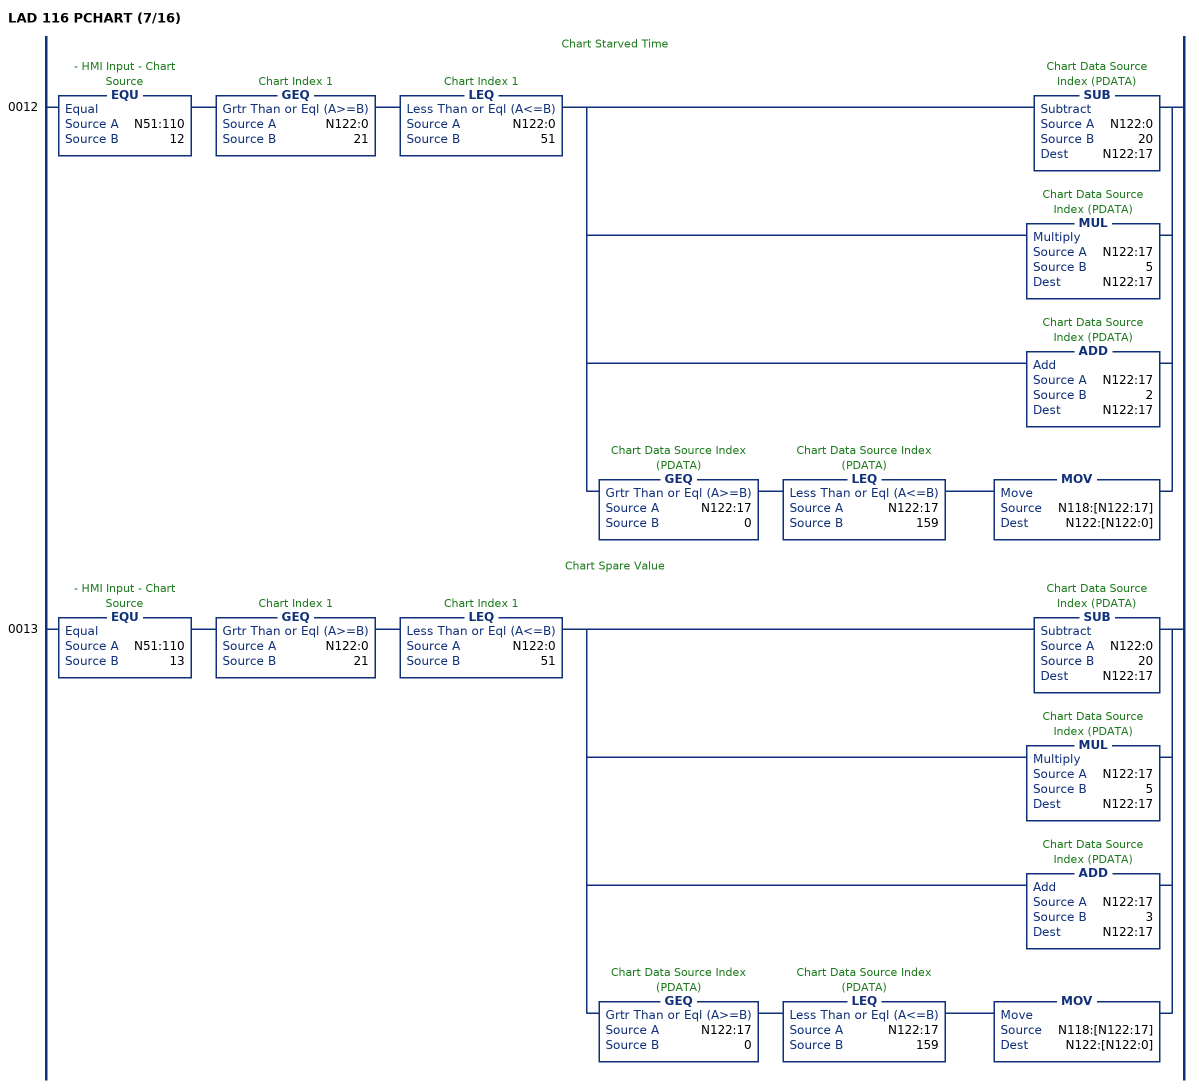
% Rung: 12 %
% Chart Starved Time %
SOR EQU N51:110 12 GEQ N122:0 21 LEQ N122:0 51 BST SUB N122:0 20 N122:17 NXB MUL N122:17 5 N122:17 NXB ADD N122:17 2 N122:17 NXB GEQ N122:17 0 LEQ N122:17 159 MOV N118:[N122:17] N122:[N122:0] BND EOR
%   N51:110  "- HMI Input - Chart Source" %
%   N122:0  "Chart Index 1" %
%   N122:17  "Chart Data Source Index (PDATA)" %
% Rung: 13 %
% Chart Spare Value %
SOR EQU N51:110 13 GEQ N122:0 21 LEQ N122:0 51 BST SUB N122:0 20 N122:17 NXB MUL N122:17 5 N122:17 NXB ADD N122:17 3 N122:17 NXB GEQ N122:17 0 LEQ N122:17 159 MOV N118:[N122:17] N122:[N122:0] BND EOR
%   N51:110  "- HMI Input - Chart Source" %
%   N122:0  "Chart Index 1" %
%   N122:17  "Chart Data Source Index (PDATA)" %

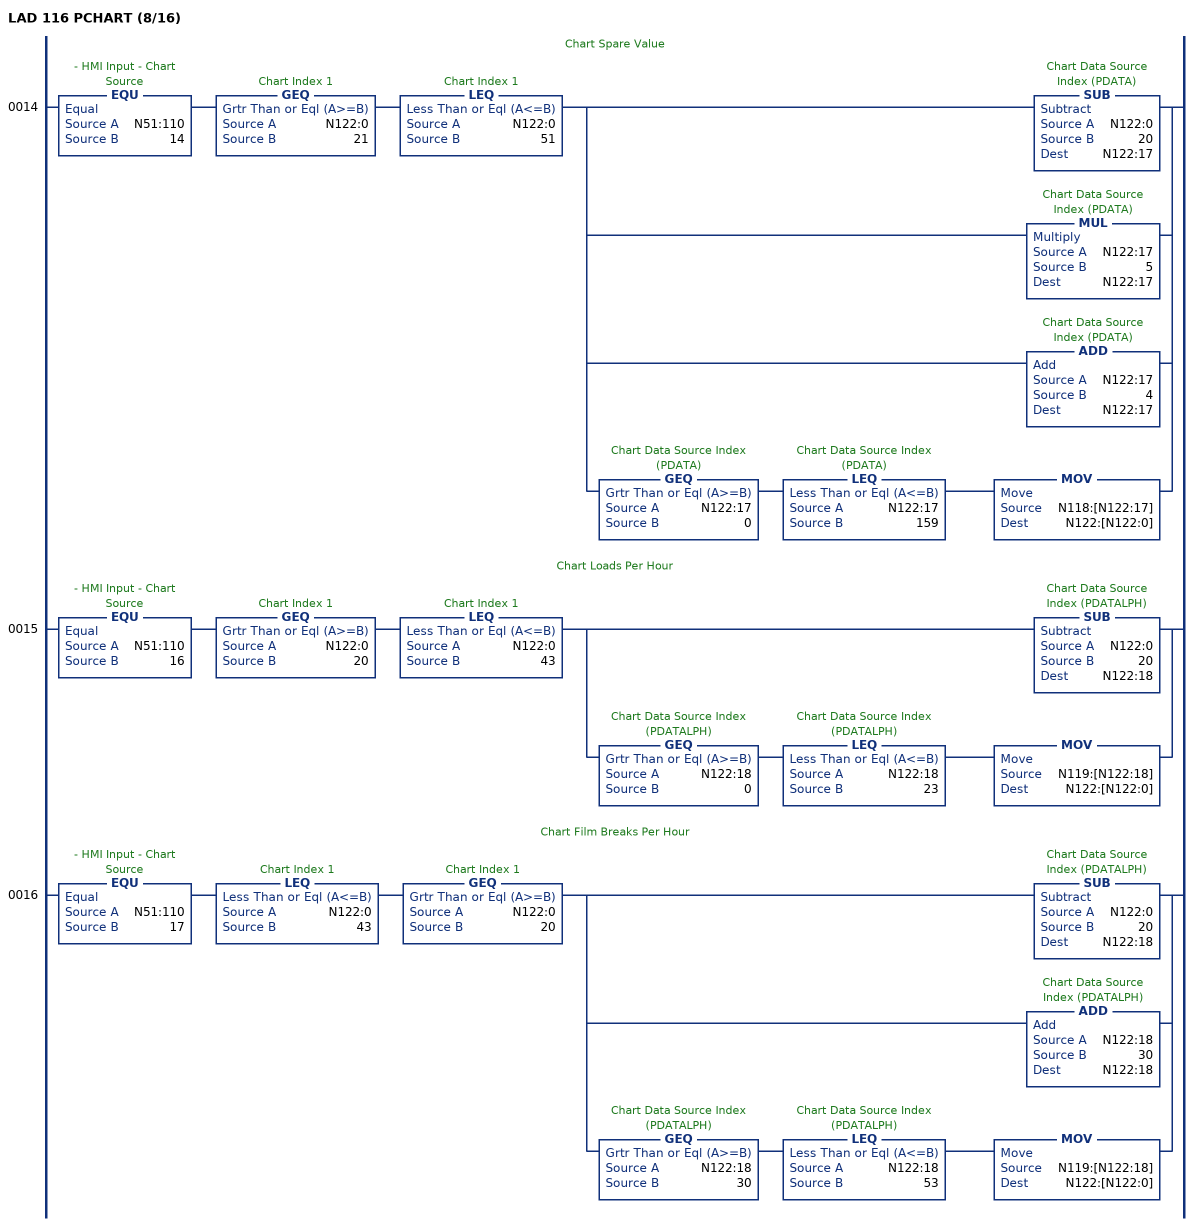
% Rung: 14 %
% Chart Spare Value %
SOR EQU N51:110 14 GEQ N122:0 21 LEQ N122:0 51 BST SUB N122:0 20 N122:17 NXB MUL N122:17 5 N122:17 NXB ADD N122:17 4 N122:17 NXB GEQ N122:17 0 LEQ N122:17 159 MOV N118:[N122:17] N122:[N122:0] BND EOR
%   N51:110  "- HMI Input - Chart Source" %
%   N122:0  "Chart Index 1" %
%   N122:17  "Chart Data Source Index (PDATA)" %
% Rung: 15 %
% Chart Loads Per Hour %
SOR EQU N51:110 16 GEQ N122:0 20 LEQ N122:0 43 BST SUB N122:0 20 N122:18 NXB GEQ N122:18 0 LEQ N122:18 23 MOV N119:[N122:18] N122:[N122:0] BND EOR
%   N51:110  "- HMI Input - Chart Source" %
%   N122:0  "Chart Index 1" %
%   N122:18  "Chart Data Source Index (PDATALPH)" %
% Rung: 16 %
% Chart Film Breaks Per Hour %
SOR EQU N51:110 17 LEQ N122:0 43 GEQ N122:0 20 BST SUB N122:0 20 N122:18 NXB ADD N122:18 30 N122:18 NXB GEQ N122:18 30 LEQ N122:18 53 MOV N119:[N122:18] N122:[N122:0] BND EOR
%   N51:110  "- HMI Input - Chart Source" %
%   N122:0  "Chart Index 1" %
%   N122:18  "Chart Data Source Index (PDATALPH)" %

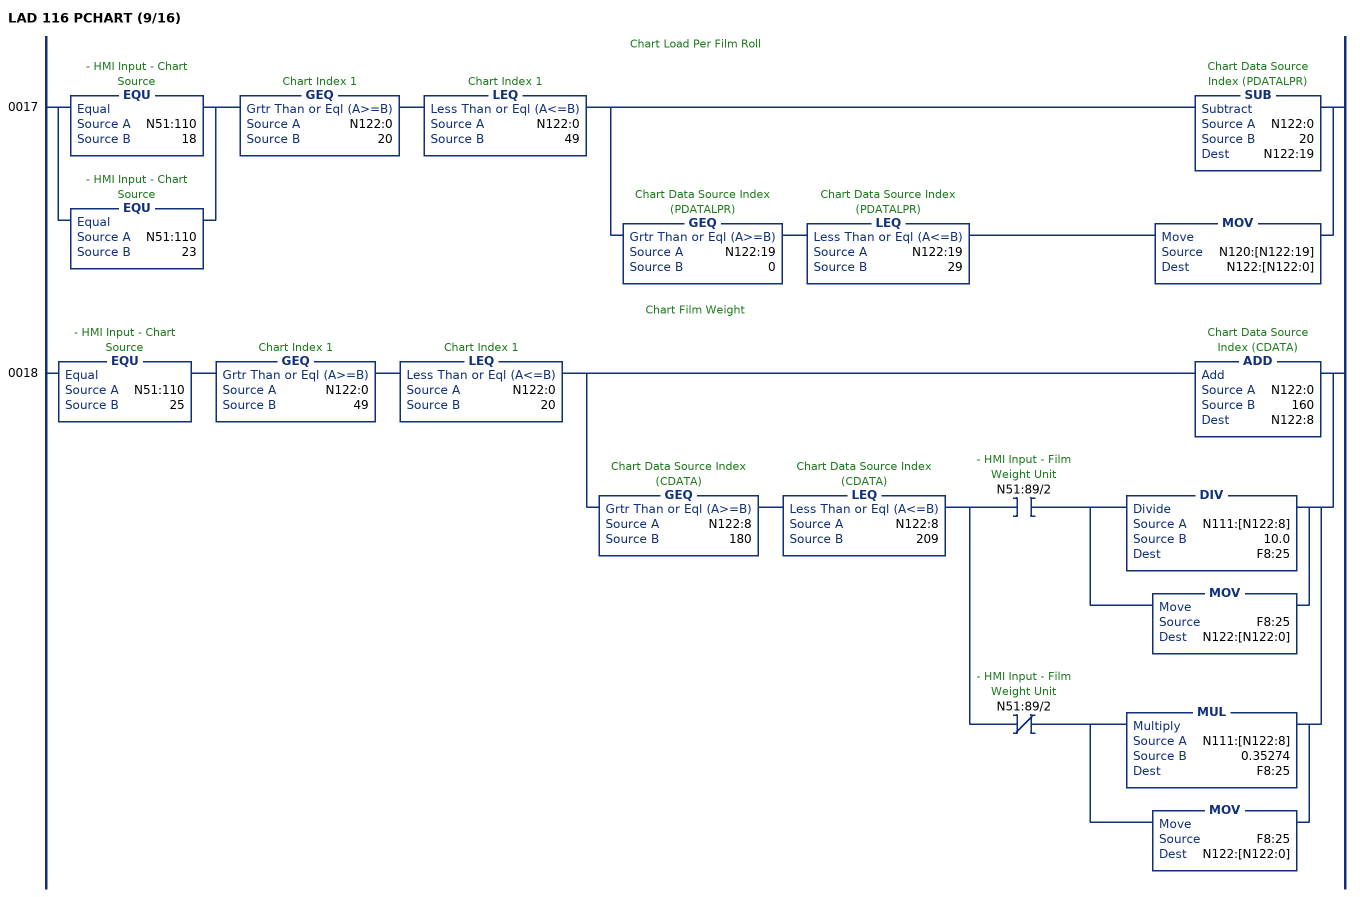
% Rung: 17 %
% Chart Load Per Film Roll %
SOR BST EQU N51:110 18 NXB EQU N51:110 23 BND GEQ N122:0 20 LEQ N122:0 49 BST SUB N122:0 20 N122:19 NXB GEQ N122:19 0 LEQ N122:19 29 MOV N120:[N122:19] N122:[N122:0] BND EOR
%   N51:110  "- HMI Input - Chart Source" %
%   N122:0  "Chart Index 1" %
%   N122:19  "Chart Data Source Index (PDATALPR)" %
% Rung: 18 %
% Chart Film Weight %
SOR EQU N51:110 25 GEQ N122:0 49 LEQ N122:0 20 BST ADD N122:0 160 N122:8 NXB GEQ N122:8 180 LEQ N122:8 209 BST XIC N51:89/2 BST DIV N111:[N122:8] 10.0 F8:25 NXB MOV F8:25 N122:[N122:0] BND NXB XIO N51:89/2 BST MUL N111:[N122:8] 0.35274 F8:25 NXB MOV F8:25 N122:[N122:0] BND BND BND EOR
%   N51:110  "- HMI Input - Chart Source" %
%   N122:0  "Chart Index 1" %
%   N122:8  "Chart Data Source Index (CDATA)" %
%   N51:89/2  "- HMI Input - Film Weight Unit" %

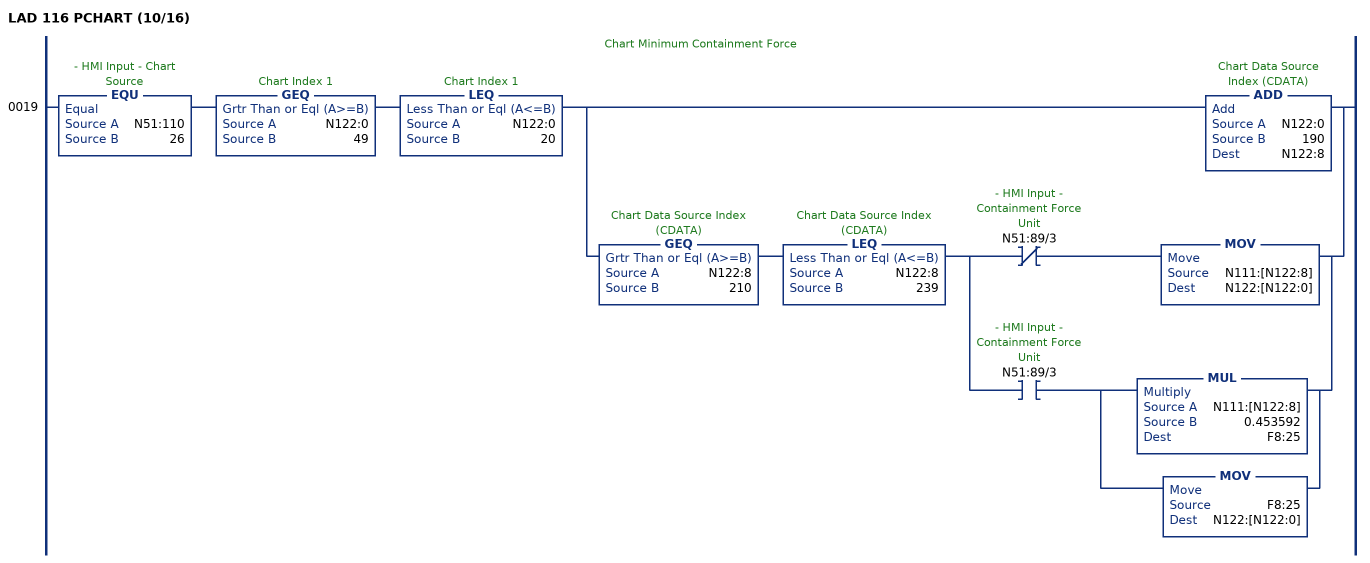
% Rung: 19 %
% Chart Minimum Containment Force %
SOR EQU N51:110 26 GEQ N122:0 49 LEQ N122:0 20 BST ADD N122:0 190 N122:8 NXB GEQ N122:8 210 LEQ N122:8 239 BST XIO N51:89/3 MOV N111:[N122:8] N122:[N122:0] NXB XIC N51:89/3 BST MUL N111:[N122:8] 0.453592 F8:25 NXB MOV F8:25 N122:[N122:0] BND BND BND EOR
%   N51:110  "- HMI Input - Chart Source" %
%   N122:0  "Chart Index 1" %
%   N122:8  "Chart Data Source Index (CDATA)" %
%   N51:89/3  "- HMI Input - Containment Force Unit" %

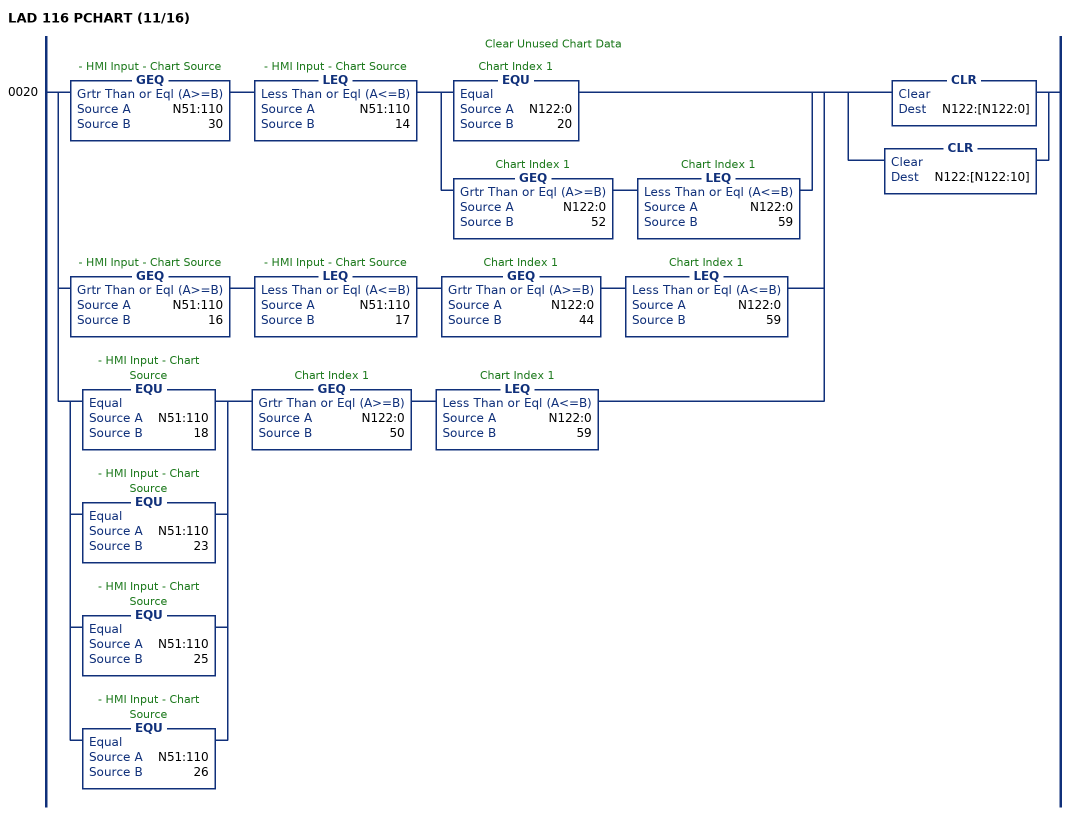
% Rung: 20 %
% Clear Unused Chart Data %
SOR BST GEQ N51:110 30 LEQ N51:110 14 BST EQU N122:0 20 NXB GEQ N122:0 52 LEQ N122:0 59 BND NXB GEQ N51:110 16 LEQ N51:110 17 GEQ N122:0 44 LEQ N122:0 59 NXB BST EQU N51:110 18 NXB EQU N51:110 23 NXB EQU N51:110 25 NXB EQU N51:110 26 BND GEQ N122:0 50 LEQ N122:0 59 BND BST CLR N122:[N122:0] NXB CLR N122:[N122:10] BND EOR
%   N51:110  "- HMI Input - Chart Source" %
%   N122:0  "Chart Index 1" %
%   N122:10  "Chart Index 2" %

